LIN {X 0,Y 524.222,Z 576.731,A -85,B 0,C 180,E1 -4783.371,E2 -4783.371} C_VEL
LIN {X 0,Y 524.644,Z 566.022,A -85,B 0,C 180,E1 -4784.886,E2 -4784.886} C_VEL
LIN {X 0,Y 525.141,Z 554.055,A -85,B 0,C 180,E1 -4786.323,E2 -4786.323} C_VEL
LIN {X 0,Y 525.695,Z 541.49,A -85,B 0,C 180,E1 -4787.606,E2 -4787.606} C_VEL
LIN {X 0,Y 526.345,Z 527.816,A -85,B 0,C 180,E1 -4788.792,E2 -4788.792} C_VEL
LIN {X 0,Y 526.961,Z 514.228,A -85,B 0,C 180,E1 -4789.781,E2 -4789.781} C_VEL
LIN {X 0,Y 527.519,Z 499.628,A -85,B 0,C 180,E1 -4790.674,E2 -4790.674} C_VEL
LIN {X 0,Y 528.182,Z 483.147,A -85,B 0,C 180,E1 -4791.492,E2 -4791.492} C_VEL
LIN {X 0,Y 528.713,Z 467.343,A -85,B 0,C 180,E1 -4792.108,E2 -4792.108} C_VEL
LIN {X 0,Y 529.094,Z 451.309,A -85,B 0,C 180,E1 -4792.579,E2 -4792.579} C_VEL
LIN {X 0,Y 529.403,Z 434.816,A -85,B 0,C 180,E1 -4792.9,E2 -4792.9} C_VEL
LIN {X 0,Y 530.91,Z 248.916,A -85,B 0,C 180,E1 -4795.546,E2 -4795.546} C_VEL
LIN {X 0,Y 528.192,Z 233.834,A -85,B 0,C 180,E1 -4795.919,E2 -4795.919} C_VEL
LIN {X 0,Y 529.034,Z 209.98,A -85,B 0,C 180,E1 -4798.169,E2 -4798.169} C_VEL
LIN {X 0,Y 524.534,Z 194.611,A -85,B 0,C 180,E1 -4799.94,E2 -4799.94} C_VEL
LIN {X 0,Y 523.914,Z 192.537,A -85,B 0,C 180,E1 -4800.201,E2 -4800.201} C_VEL
LIN {X 0,Y 523.939,Z 192.528,A -85,B 0,C 180,E1 -4803.364,E2 -4803.364} C_VEL
LIN {X 0,Y 523.896,Z 192.537,A -85,B 0,C 180,E1 -4806.4,E2 -4806.4} C_VEL
LIN {X 0,Y 523.917,Z 192.54,A -85,B 0,C 180,E1 -4809.085,E2 -4809.085} C_VEL
LIN {X 0,Y 523.936,Z 192.53,A -85,B 0,C 180,E1 -4812.12,E2 -4812.12} C_VEL
LIN {X 0,Y 523.936,Z 192.531,A -85,B 0,C 180,E1 -4815.311,E2 -4815.311} C_VEL
LIN {X 0,Y 523.95,Z 192.533,A -85,B 0,C 180,E1 -4818.69,E2 -4818.69} C_VEL
LIN {X 0,Y 523.911,Z 192.533,A -85,B 0,C 180,E1 -4821.898,E2 -4821.898} C_VEL
LIN {X 0,Y 523.92,Z 192.537,A -85,B 0,C 180,E1 -4824.911,E2 -4824.911} C_VEL
LIN {X 0,Y 523.931,Z 192.526,A -85,B 0,C 180,E1 -4827.68,E2 -4827.68} C_VEL
LIN {X 0,Y 523.949,Z 192.534,A -85,B 0,C 180,E1 -4830.677,E2 -4830.677} C_VEL
LIN {X 0,Y 523.969,Z 192.519,A -85,B 0,C 180,E1 -4833.728,E2 -4833.728} C_VEL
LIN {X 0,Y 523.909,Z 192.534,A -85,B 0,C 180,E1 -4836.27,E2 -4836.27} C_VEL
LIN {X 0,Y 523.941,Z 192.531,A -85,B 0,C 180,E1 -4838.767,E2 -4838.767} C_VEL
LIN {X 0,Y 523.936,Z 192.524,A -85,B 0,C 180,E1 -4841.22,E2 -4841.22} C_VEL
LIN {X 0,Y 523.924,Z 192.53,A -85,B 0,C 180,E1 -4843.639,E2 -4843.639} C_VEL
LIN {X 0,Y 523.934,Z 192.531,A -85,B 0,C 180,E1 -4846.028,E2 -4846.028} C_VEL
LIN {X 0,Y 524.009,Z 192.516,A -85,B 0,C 180,E1 -4848.394,E2 -4848.394} C_VEL
LIN {X 0,Y 523.986,Z 192.522,A -85,B 0,C 180,E1 -4851.516,E2 -4851.516} C_VEL
LIN {X 0,Y 524.032,Z 192.519,A -85,B 0,C 180,E1 -4853.841,E2 -4853.841} C_VEL
LIN {X 0,Y 524.067,Z 192.501,A -85,B 0,C 180,E1 -4856.925,E2 -4856.925} C_VEL
LIN {X 0,Y 524.109,Z 192.509,A -85,B 0,C 180,E1 -4860,E2 -4860} C_VEL
LIN {X 0,Y 524.068,Z 192.511,A -85,B 0,C 180,E1 -4863.075,E2 -4863.075} C_VEL
LIN {X 0,Y 524.041,Z 192.518,A -85,B 0,C 180,E1 -4866.159,E2 -4866.159} C_VEL
LIN {X 0,Y 523.997,Z 192.525,A -85,B 0,C 180,E1 -4868.484,E2 -4868.484} C_VEL
LIN {X 0,Y 523.999,Z 192.521,A -85,B 0,C 180,E1 -4871.739,E2 -4871.739} C_VEL
LIN {X 0,Y 523.99,Z 192.522,A -85,B 0,C 180,E1 -4875.052,E2 -4875.052} C_VEL
LIN {X 0,Y 523.962,Z 192.527,A -85,B 0,C 180,E1 -4877.969,E2 -4877.969} C_VEL
LIN {X 0,Y 523.969,Z 192.526,A -85,B 0,C 180,E1 -4880.41,E2 -4880.41} C_VEL
LIN {X 0,Y 523.914,Z 192.531,A -85,B 0,C 180,E1 -4882.893,E2 -4882.893} C_VEL
LIN {X 0,Y 523.95,Z 192.525,A -85,B 0,C 180,E1 -4885.419,E2 -4885.419} C_VEL
LIN {X 0,Y 523.968,Z 192.531,A -85,B 0,C 180,E1 -4887.999,E2 -4887.999} C_VEL
LIN {X 0,Y 523.947,Z 192.525,A -85,B 0,C 180,E1 -4890.856,E2 -4890.856} C_VEL
LIN {X 0,Y 523.959,Z 192.532,A -85,B 0,C 180,E1 -4893.735,E2 -4893.735} C_VEL
LIN {X 0,Y 523.92,Z 192.53,A -85,B 0,C 180,E1 -4896.404,E2 -4896.404} C_VEL
LIN {X 0,Y 523.917,Z 192.529,A -85,B 0,C 180,E1 -4899.085,E2 -4899.085} C_VEL
LIN {X 0,Y 523.952,Z 192.527,A -85,B 0,C 180,E1 -4902.119,E2 -4902.119} C_VEL
LIN {X 0,Y 523.944,Z 192.531,A -85,B 0,C 180,E1 -4905.31,E2 -4905.31} C_VEL
LIN {X 0,Y 523.916,Z 192.533,A -85,B 0,C 180,E1 -4906.916,E2 -4906.916} C_VEL
LIN {X 0,Y 523.249,Z 192.62,A -85,B 0,C 180,E1 -4907.558,E2 -4907.558} C_VEL
LIN {X 0,Y 520.407,Z 192.971,A -85,B 0,C 180,E1 -4908.599,E2 -4908.599} C_VEL
LIN {X 0,Y 518.003,Z 193.272,A -85,B 0,C 180,E1 -4909.438,E2 -4909.438} C_VEL
LIN {X 0,Y 516.966,Z 193.398,A -85,B 0,C 180,E1 -4910.086,E2 -4910.086} C_VEL
LIN {X 0,Y 516.879,Z 193.408,A -85,B 0,C 180,E1 -4910.305,E2 -4910.305} C_VEL
LIN {X 0,Y 516.875,Z 193.412,A -85,B 0,C 180,E1 -4913.343,E2 -4913.343} C_VEL
LIN {X 0,Y 516.909,Z 193.406,A -85,B 0,C 180,E1 -4916.121,E2 -4916.121} C_VEL
LIN {X 0,Y 516.89,Z 193.408,A -85,B 0,C 180,E1 -4918.936,E2 -4918.936} C_VEL
LIN {X 0,Y 516.917,Z 193.406,A -85,B 0,C 180,E1 -4921.585,E2 -4921.585} C_VEL
LIN {X 0,Y 516.931,Z 193.402,A -85,B 0,C 180,E1 -4924.211,E2 -4924.211} C_VEL
LIN {X 0,Y 516.865,Z 193.411,A -85,B 0,C 180,E1 -4926.776,E2 -4926.776} C_VEL
LIN {X 0,Y 516.939,Z 193.397,A -85,B 0,C 180,E1 -4929.732,E2 -4929.732} C_VEL
LIN {X 0,Y 516.906,Z 193.405,A -85,B 0,C 180,E1 -4932.595,E2 -4932.595} C_VEL
LIN {X 0,Y 516.942,Z 193.402,A -85,B 0,C 180,E1 -4935.03,E2 -4935.03} C_VEL
LIN {X 0,Y 516.965,Z 193.4,A -85,B 0,C 180,E1 -4938.234,E2 -4938.234} C_VEL
LIN {X 0,Y 516.968,Z 193.402,A -85,B 0,C 180,E1 -4941.4,E2 -4941.4} C_VEL
LIN {X 0,Y 517.026,Z 193.393,A -85,B 0,C 180,E1 -4944.54,E2 -4944.54} C_VEL
LIN {X 0,Y 517.047,Z 193.434,A -85,B 0,C 180,E1 -4947.979,E2 -4947.979} C_VEL
LIN {X 0,Y 520.935,Z 207.525,A -85,B 0,C 180,E1 -4949.764,E2 -4949.764} C_VEL
LIN {X 0,Y 522.633,Z 212.295,A -85,B 0,C 180,E1 -4949.929,E2 -4949.929} C_VEL
LIN {X 0,Y 524.563,Z 222.327,A -85,B 0,C 180,E1 -4950.184,E2 -4950.184} C_VEL
LIN {X 0,Y 522.855,Z 413.311,A -85,B 0,C 180,E1 -4952.961,E2 -4952.961} C_VEL
LIN {X 0,Y 522.525,Z 429.48,A -85,B 0,C 180,E1 -4953.349,E2 -4953.349} C_VEL
LIN {X 0,Y 521.977,Z 445.854,A -85,B 0,C 180,E1 -4953.898,E2 -4953.898} C_VEL
LIN {X 0,Y 521.414,Z 460.885,A -85,B 0,C 180,E1 -4954.555,E2 -4954.555} C_VEL
LIN {X 0,Y 520.78,Z 476.68,A -85,B 0,C 180,E1 -4955.42,E2 -4955.42} C_VEL
LIN {X 0,Y 520.083,Z 491.283,A -85,B 0,C 180,E1 -4956.401,E2 -4956.401} C_VEL
LIN {X 0,Y 519.44,Z 504.752,A -85,B 0,C 180,E1 -4957.482,E2 -4957.482} C_VEL
LIN {X 0,Y 518.713,Z 518.29,A -85,B 0,C 180,E1 -4958.767,E2 -4958.767} C_VEL
LIN {X 0,Y 518.081,Z 530.647,A -85,B 0,C 180,E1 -4960.157,E2 -4960.157} C_VEL
LIN {X 0,Y 517.589,Z 541.233,A -85,B 0,C 180,E1 -4961.553,E2 -4961.553} C_VEL
LIN {X 0,Y 517.153,Z 551.508,A -85,B 0,C 180,E1 -4963.157,E2 -4963.157} C_VEL
LIN {X 0,Y 516.805,Z 560.149,A -85,B 0,C 180,E1 -4964.772,E2 -4964.772} C_VEL
LIN {X 0,Y 516.566,Z 566.583,A -85,B 0,C 180,E1 -4966.195,E2 -4966.195} C_VEL
LIN {X 0,Y 516.446,Z 572.319,A -85,B 0,C 180,E1 -4967.715,E2 -4967.715} C_VEL
LIN {X 0,Y 516.32,Z 577.625,A -85,B 0,C 180,E1 -4969.48,E2 -4969.48} C_VEL
LIN {X 0,Y 516.228,Z 580.6,A -85,B 0,C 180,E1 -4970.73,E2 -4970.73} C_VEL
LIN {X 0,Y 516.174,Z 583.527,A -85,B 0,C 180,E1 -4972.41,E2 -4972.41} C_VEL
LIN {X 0,Y 516.138,Z 585.436,A -85,B 0,C 180,E1 -4974.174,E2 -4974.174} C_VEL
LIN {X 0,Y 516.146,Z 586.138,A -85,B 0,C 180,E1 -4976.016,E2 -4976.016} C_VEL
LIN {X 0,Y 516.168,Z 585.538,A -85,B 0,C 180,E1 -4977.746,E2 -4977.746} C_VEL
LIN {X 0,Y 516.193,Z 583.95,A -85,B 0,C 180,E1 -4979.383,E2 -4979.383} C_VEL
LIN {X 0,Y 516.235,Z 581.052,A -85,B 0,C 180,E1 -4981.153,E2 -4981.153} C_VEL
LIN {X 0,Y 516.314,Z 578.077,A -85,B 0,C 180,E1 -4982.442,E2 -4982.442} C_VEL
LIN {X 0,Y 516.384,Z 573.835,A -85,B 0,C 180,E1 -4983.918,E2 -4983.918} C_VEL
LIN {X 0,Y 516.54,Z 568.152,A -85,B 0,C 180,E1 -4985.508,E2 -4985.508} C_VEL
LIN {X 0,Y 516.737,Z 560.548,A -85,B 0,C 180,E1 -4987.245,E2 -4987.245} C_VEL
LIN {X 0,Y 517.046,Z 552.873,A -85,B 0,C 180,E1 -4988.7,E2 -4988.7} C_VEL
LIN {X 0,Y 517.441,Z 543.71,A -85,B 0,C 180,E1 -4990.176,E2 -4990.176} C_VEL
LIN {X 0,Y 517.976,Z 532.31,A -85,B 0,C 180,E1 -4991.734,E2 -4991.734} C_VEL
LIN {X 0,Y 518.636,Z 519.838,A -85,B 0,C 180,E1 -4993.168,E2 -4993.168} C_VEL
LIN {X 0,Y 519.267,Z 507.368,A -85,B 0,C 180,E1 -4994.388,E2 -4994.388} C_VEL
LIN {X 0,Y 520.016,Z 492.6,A -85,B 0,C 180,E1 -4995.6,E2 -4995.6} C_VEL
LIN {X 0,Y 520.798,Z 476.677,A -85,B 0,C 180,E1 -4996.675,E2 -4996.675} C_VEL
LIN {X 0,Y 521.453,Z 460.886,A -85,B 0,C 180,E1 -4997.538,E2 -4997.538} C_VEL
LIN {X 0,Y 522.01,Z 445.593,A -85,B 0,C 180,E1 -4998.204,E2 -4998.204} C_VEL
LIN {X 0,Y 522.498,Z 429.104,A -85,B 0,C 180,E1 -4998.754,E2 -4998.754} C_VEL
LIN {X 0,Y 522.873,Z 412.973,A -85,B 0,C 180,E1 -4999.135,E2 -4999.135} C_VEL
LIN {X 0,Y 524.555,Z 221.705,A -85,B 0,C 180,E1 -5001.919,E2 -5001.919} C_VEL
LIN {X 0,Y 522.049,Z 210.335,A -85,B 0,C 180,E1 -5002.227,E2 -5002.227} C_VEL
LIN {X 0,Y 520.799,Z 207.327,A -85,B 0,C 180,E1 -5002.365,E2 -5002.365} C_VEL
LIN {X 0,Y 516.875,Z 193.415,A -85,B 0,C 180,E1 -5004.19,E2 -5004.19} C_VEL
LIN {X 0,Y 516.874,Z 193.417,A -85,B 0,C 180,E1 -5007.052,E2 -5007.052} C_VEL
LIN {X 0,Y 516.875,Z 193.413,A -85,B 0,C 180,E1 -5009.795,E2 -5009.795} C_VEL
LIN {X 0,Y 516.883,Z 193.412,A -85,B 0,C 180,E1 -5012.465,E2 -5012.465} C_VEL
LIN {X 0,Y 516.866,Z 193.412,A -85,B 0,C 180,E1 -5015.645,E2 -5015.645} C_VEL
LIN {X 0,Y 516.877,Z 193.41,A -85,B 0,C 180,E1 -5018.462,E2 -5018.462} C_VEL
LIN {X 0,Y 516.892,Z 193.411,A -85,B 0,C 180,E1 -5020.955,E2 -5020.955} C_VEL
LIN {X 0,Y 516.897,Z 193.407,A -85,B 0,C 180,E1 -5023.41,E2 -5023.41} C_VEL
LIN {X 0,Y 516.885,Z 193.409,A -85,B 0,C 180,E1 -5025.833,E2 -5025.833} C_VEL
LIN {X 0,Y 516.958,Z 193.399,A -85,B 0,C 180,E1 -5028.234,E2 -5028.234} C_VEL
LIN {X 0,Y 516.95,Z 193.4,A -85,B 0,C 180,E1 -5031.399,E2 -5031.399} C_VEL
LIN {X 0,Y 516.994,Z 193.394,A -85,B 0,C 180,E1 -5033.757,E2 -5033.757} C_VEL
LIN {X 0,Y 517.006,Z 193.395,A -85,B 0,C 180,E1 -5036.883,E2 -5036.883} C_VEL
LIN {X 0,Y 517.076,Z 193.389,A -85,B 0,C 180,E1 -5040,E2 -5040} C_VEL
LIN {X 0,Y 517.006,Z 193.391,A -85,B 0,C 180,E1 -5043.117,E2 -5043.117} C_VEL
LIN {X 0,Y 517.002,Z 193.4,A -85,B 0,C 180,E1 -5046.243,E2 -5046.243} C_VEL
LIN {X 0,Y 516.948,Z 193.401,A -85,B 0,C 180,E1 -5049.389,E2 -5049.389} C_VEL
LIN {X 0,Y 516.945,Z 193.404,A -85,B 0,C 180,E1 -5051.808,E2 -5051.808} C_VEL
LIN {X 0,Y 516.937,Z 193.402,A -85,B 0,C 180,E1 -5055.147,E2 -5055.147} C_VEL
LIN {X 0,Y 516.919,Z 193.406,A -85,B 0,C 180,E1 -5058.222,E2 -5058.222} C_VEL
LIN {X 0,Y 516.906,Z 193.406,A -85,B 0,C 180,E1 -5060.702,E2 -5060.702} C_VEL
LIN {X 0,Y 516.905,Z 193.409,A -85,B 0,C 180,E1 -5064.072,E2 -5064.072} C_VEL
LIN {X 0,Y 516.923,Z 193.402,A -85,B 0,C 180,E1 -5066.658,E2 -5066.658} C_VEL
LIN {X 0,Y 516.905,Z 193.412,A -85,B 0,C 180,E1 -5069.524,E2 -5069.524} C_VEL
LIN {X 0,Y 516.895,Z 193.408,A -85,B 0,C 180,E1 -5072.545,E2 -5072.545} C_VEL
LIN {X 0,Y 516.865,Z 193.42,A -85,B 0,C 180,E1 -5075.331,E2 -5075.331} C_VEL
LIN {X 0,Y 516.875,Z 193.413,A -85,B 0,C 180,E1 -5077.944,E2 -5077.944} C_VEL
LIN {X 0,Y 516.879,Z 193.413,A -85,B 0,C 180,E1 -5080.742,E2 -5080.742} C_VEL
LIN {X 0,Y 516.878,Z 193.415,A -85,B 0,C 180,E1 -5082.832,E2 -5082.832} C_VEL
LIN {X 0,Y 516.918,Z 193.414,A -85,B 0,C 180,E1 -5085.011,E2 -5085.011} C_VEL
LIN {X 0,Y 516.908,Z 193.409,A -85,B 0,C 180,E1 -5088.399,E2 -5088.399} C_VEL
LIN {X 0,Y 516.877,Z 193.414,A -85,B 0,C 180,E1 -5091.285,E2 -5091.285} C_VEL
LIN {X 0,Y 516.866,Z 193.414,A -85,B 0,C 180,E1 -5094.22,E2 -5094.22} C_VEL
LIN {X 0,Y 516.891,Z 193.416,A -85,B 0,C 180,E1 -5097.053,E2 -5097.053} C_VEL
LIN {X 0,Y 516.916,Z 193.581,A -85,B 0,C 180,E1 -5099.516,E2 -5099.516} C_VEL
LIN {X 0,Y 522.209,Z 211.448,A -85,B 0,C 180,E1 -5101.62,E2 -5101.62} C_VEL
LIN {X 0,Y 521.508,Z 233.414,A -85,B 0,C 180,E1 -5103.727,E2 -5103.727} C_VEL
LIN {X 0,Y 524.478,Z 250.636,A -85,B 0,C 180,E1 -5104.151,E2 -5104.151} C_VEL
LIN {X 0,Y 522.789,Z 438.701,A -85,B 0,C 180,E1 -5106.872,E2 -5106.872} C_VEL
LIN {X 0,Y 522.446,Z 454.476,A -85,B 0,C 180,E1 -5107.222,E2 -5107.222} C_VEL
LIN {X 0,Y 522.001,Z 469.792,A -85,B 0,C 180,E1 -5107.698,E2 -5107.698} C_VEL
LIN {X 0,Y 521.425,Z 484.424,A -85,B 0,C 180,E1 -5108.294,E2 -5108.294} C_VEL
LIN {X 0,Y 520.852,Z 499.253,A -85,B 0,C 180,E1 -5109.049,E2 -5109.049} C_VEL
LIN {X 0,Y 520.249,Z 512.438,A -85,B 0,C 180,E1 -5109.851,E2 -5109.851} C_VEL
LIN {X 0,Y 519.508,Z 527.483,A -85,B 0,C 180,E1 -5110.952,E2 -5110.952} C_VEL
LIN {X 0,Y 518.864,Z 540.105,A -85,B 0,C 180,E1 -5112.053,E2 -5112.053} C_VEL
LIN {X 0,Y 518.276,Z 551.972,A -85,B 0,C 180,E1 -5113.253,E2 -5113.253} C_VEL
LIN {X 0,Y 517.734,Z 563.934,A -85,B 0,C 180,E1 -5114.666,E2 -5114.666} C_VEL
LIN {X 0,Y 517.265,Z 575.232,A -85,B 0,C 180,E1 -5116.245,E2 -5116.245} C_VEL
LIN {X 0,Y 516.933,Z 584.758,A -85,B 0,C 180,E1 -5117.835,E2 -5117.835} C_VEL
LIN {X 0,Y 516.672,Z 592.73,A -85,B 0,C 180,E1 -5119.419,E2 -5119.419} C_VEL
LIN {X 0,Y 516.468,Z 599.381,A -85,B 0,C 180,E1 -5120.997,E2 -5120.997} C_VEL
LIN {X 0,Y 516.371,Z 604.775,A -85,B 0,C 180,E1 -5122.571,E2 -5122.571} C_VEL
LIN {X 0,Y 516.319,Z 608.108,A -85,B 0,C 180,E1 -5123.749,E2 -5123.749} C_VEL
LIN {X 0,Y 516.225,Z 611.529,A -85,B 0,C 180,E1 -5125.315,E2 -5125.315} C_VEL
LIN {X 0,Y 516.267,Z 614.018,A -85,B 0,C 180,E1 -5126.879,E2 -5126.879} C_VEL
LIN {X 0,Y 516.186,Z 615.418,A -85,B 0,C 180,E1 -5128.44,E2 -5128.44} C_VEL
LIN {X 0,Y 516.149,Z 615.946,A -85,B 0,C 180,E1 -5130,E2 -5130} C_VEL
LIN {X 0,Y 516.186,Z 615.418,A -85,B 0,C 180,E1 -5131.561,E2 -5131.561} C_VEL
LIN {X 0,Y 516.267,Z 614.017,A -85,B 0,C 180,E1 -5133.122,E2 -5133.122} C_VEL
LIN {X 0,Y 516.225,Z 611.53,A -85,B 0,C 180,E1 -5134.686,E2 -5134.686} C_VEL
LIN {X 0,Y 516.368,Z 607.414,A -85,B 0,C 180,E1 -5136.507,E2 -5136.507} C_VEL
LIN {X 0,Y 516.418,Z 602.265,A -85,B 0,C 180,E1 -5138.216,E2 -5138.216} C_VEL
LIN {X 0,Y 516.591,Z 594.571,A -85,B 0,C 180,E1 -5140.187,E2 -5140.187} C_VEL
LIN {X 0,Y 516.904,Z 585.889,A -85,B 0,C 180,E1 -5141.967,E2 -5141.967} C_VEL
LIN {X 0,Y 517.203,Z 576.513,A -85,B 0,C 180,E1 -5143.556,E2 -5143.556} C_VEL
LIN {X 0,Y 517.635,Z 566.866,A -85,B 0,C 180,E1 -5144.949,E2 -5144.949} C_VEL
LIN {X 0,Y 518.134,Z 555.623,A -85,B 0,C 180,E1 -5146.347,E2 -5146.347} C_VEL
LIN {X 0,Y 518.751,Z 543.377,A -85,B 0,C 180,E1 -5147.646,E2 -5147.646} C_VEL
LIN {X 0,Y 519.397,Z 530.405,A -85,B 0,C 180,E1 -5148.812,E2 -5148.812} C_VEL
LIN {X 0,Y 520.043,Z 516.853,A -85,B 0,C 180,E1 -5149.849,E2 -5149.849} C_VEL
LIN {X 0,Y 520.639,Z 502.921,A -85,B 0,C 180,E1 -5150.753,E2 -5150.753} C_VEL
LIN {X 0,Y 521.415,Z 487.208,A -85,B 0,C 180,E1 -5151.584,E2 -5151.584} C_VEL
LIN {X 0,Y 521.956,Z 471.272,A -85,B 0,C 180,E1 -5152.253,E2 -5152.253} C_VEL
LIN {X 0,Y 522.403,Z 455.599,A -85,B 0,C 180,E1 -5152.754,E2 -5152.754} C_VEL
LIN {X 0,Y 522.791,Z 438.955,A -85,B 0,C 180,E1 -5153.128,E2 -5153.128} C_VEL
LIN {X 0,Y 524.44,Z 249.524,A -85,B 0,C 180,E1 -5155.872,E2 -5155.872} C_VEL
LIN {X 0,Y 521.559,Z 233.731,A -85,B 0,C 180,E1 -5156.265,E2 -5156.265} C_VEL
LIN {X 0,Y 522.325,Z 211.669,A -85,B 0,C 180,E1 -5158.379,E2 -5158.379} C_VEL
LIN {X 0,Y 516.901,Z 193.409,A -85,B 0,C 180,E1 -5160.542,E2 -5160.542} C_VEL
LIN {X 0,Y 516.892,Z 193.401,A -85,B 0,C 180,E1 -5162.947,E2 -5162.947} C_VEL
LIN {X 0,Y 516.865,Z 193.415,A -85,B 0,C 180,E1 -5165.781,E2 -5165.781} C_VEL
LIN {X 0,Y 516.877,Z 193.414,A -85,B 0,C 180,E1 -5168.716,E2 -5168.716} C_VEL
LIN {X 0,Y 516.899,Z 193.408,A -85,B 0,C 180,E1 -5171.776,E2 -5171.776} C_VEL
LIN {X 0,Y 516.892,Z 193.412,A -85,B 0,C 180,E1 -5175.007,E2 -5175.007} C_VEL
LIN {X 0,Y 516.906,Z 193.408,A -85,B 0,C 180,E1 -5178.399,E2 -5178.399} C_VEL
LIN {X 0,Y 516.874,Z 193.414,A -85,B 0,C 180,E1 -5181.284,E2 -5181.284} C_VEL
LIN {X 0,Y 516.867,Z 193.406,A -85,B 0,C 180,E1 -5184.22,E2 -5184.22} C_VEL
LIN {X 0,Y 516.878,Z 193.41,A -85,B 0,C 180,E1 -5187.052,E2 -5187.052} C_VEL
LIN {X 0,Y 516.888,Z 193.406,A -85,B 0,C 180,E1 -5189.796,E2 -5189.796} C_VEL
LIN {X 0,Y 516.92,Z 193.409,A -85,B 0,C 180,E1 -5192.467,E2 -5192.467} C_VEL
LIN {X 0,Y 516.869,Z 193.412,A -85,B 0,C 180,E1 -5195.07,E2 -5195.07} C_VEL
LIN {X 0,Y 516.865,Z 193.411,A -85,B 0,C 180,E1 -5197.621,E2 -5197.621} C_VEL
LIN {X 0,Y 516.926,Z 193.4,A -85,B 0,C 180,E1 -5200.13,E2 -5200.13} C_VEL
LIN {X 0,Y 516.893,Z 193.41,A -85,B 0,C 180,E1 -5202.595,E2 -5202.595} C_VEL
LIN {X 0,Y 516.939,Z 193.402,A -85,B 0,C 180,E1 -5205.03,E2 -5205.03} C_VEL
LIN {X 0,Y 516.962,Z 193.393,A -85,B 0,C 180,E1 -5208.234,E2 -5208.234} C_VEL
LIN {X 0,Y 516.954,Z 193.398,A -85,B 0,C 180,E1 -5211.399,E2 -5211.399} C_VEL
LIN {X 0,Y 516.998,Z 193.394,A -85,B 0,C 180,E1 -5213.757,E2 -5213.757} C_VEL
LIN {X 0,Y 517.008,Z 193.38,A -85,B 0,C 180,E1 -5216.883,E2 -5216.883} C_VEL
LIN {X 0,Y 517.08,Z 193.384,A -85,B 0,C 180,E1 -5220,E2 -5220} C_VEL
LIN {X 0,Y 517.008,Z 193.391,A -85,B 0,C 180,E1 -5223.117,E2 -5223.117} C_VEL
LIN {X 0,Y 517.005,Z 193.395,A -85,B 0,C 180,E1 -5226.243,E2 -5226.243} C_VEL
LIN {X 0,Y 516.942,Z 193.401,A -85,B 0,C 180,E1 -5229.389,E2 -5229.389} C_VEL
LIN {X 0,Y 516.949,Z 193.399,A -85,B 0,C 180,E1 -5231.807,E2 -5231.807} C_VEL
LIN {X 0,Y 516.941,Z 193.4,A -85,B 0,C 180,E1 -5235.146,E2 -5235.146} C_VEL
LIN {X 0,Y 516.923,Z 193.4,A -85,B 0,C 180,E1 -5238.222,E2 -5238.222} C_VEL
LIN {X 0,Y 516.909,Z 193.404,A -85,B 0,C 180,E1 -5240.702,E2 -5240.702} C_VEL
LIN {X 0,Y 516.909,Z 193.405,A -85,B 0,C 180,E1 -5244.072,E2 -5244.072} C_VEL
LIN {X 0,Y 516.924,Z 193.4,A -85,B 0,C 180,E1 -5246.658,E2 -5246.658} C_VEL
LIN {X 0,Y 516.917,Z 193.409,A -85,B 0,C 180,E1 -5249.526,E2 -5249.526} C_VEL
LIN {X 0,Y 516.895,Z 193.402,A -85,B 0,C 180,E1 -5252.544,E2 -5252.544} C_VEL
LIN {X 0,Y 516.881,Z 193.412,A -85,B 0,C 180,E1 -5255.332,E2 -5255.332} C_VEL
LIN {X 0,Y 516.878,Z 193.408,A -85,B 0,C 180,E1 -5257.943,E2 -5257.943} C_VEL
LIN {X 0,Y 516.882,Z 193.408,A -85,B 0,C 180,E1 -5260.742,E2 -5260.742} C_VEL
LIN {X 0,Y 516.88,Z 193.407,A -85,B 0,C 180,E1 -5262.832,E2 -5262.832} C_VEL
LIN {X 0,Y 516.88,Z 193.41,A -85,B 0,C 180,E1 -5266.097,E2 -5266.097} C_VEL
LIN {X 0,Y 516.911,Z 193.401,A -85,B 0,C 180,E1 -5268.399,E2 -5268.399} C_VEL
LIN {X 0,Y 516.879,Z 193.408,A -85,B 0,C 180,E1 -5270.305,E2 -5270.305} C_VEL
LIN {X 0,Y 516.208,Z 193.495,A -85,B 0,C 180,E1 -5270.956,E2 -5270.956} C_VEL
LIN {X 0,Y 513.36,Z 193.851,A -85,B 0,C 180,E1 -5272.011,E2 -5272.011} C_VEL
LIN {X 0,Y 510.95,Z 194.152,A -85,B 0,C 180,E1 -5272.861,E2 -5272.861} C_VEL
LIN {X 0,Y 509.908,Z 194.278,A -85,B 0,C 180,E1 -5273.518,E2 -5273.518} C_VEL
LIN {X 0,Y 509.819,Z 194.287,A -85,B 0,C 180,E1 -5273.74,E2 -5273.74} C_VEL
LIN {X 0,Y 509.859,Z 194.284,A -85,B 0,C 180,E1 -5276.539,E2 -5276.539} C_VEL
LIN {X 0,Y 509.844,Z 194.289,A -85,B 0,C 180,E1 -5279.334,E2 -5279.334} C_VEL
LIN {X 0,Y 509.891,Z 194.277,A -85,B 0,C 180,E1 -5282.055,E2 -5282.055} C_VEL
LIN {X 0,Y 509.875,Z 194.284,A -85,B 0,C 180,E1 -5284.704,E2 -5284.704} C_VEL
LIN {X 0,Y 509.826,Z 194.293,A -85,B 0,C 180,E1 -5287.458,E2 -5287.458} C_VEL
LIN {X 0,Y 509.916,Z 194.271,A -85,B 0,C 180,E1 -5289.845,E2 -5289.845} C_VEL
LIN {X 0,Y 509.873,Z 194.29,A -85,B 0,C 180,E1 -5293.174,E2 -5293.174} C_VEL
LIN {X 0,Y 509.863,Z 194.275,A -85,B 0,C 180,E1 -5295.634,E2 -5295.634} C_VEL
LIN {X 0,Y 509.913,Z 194.283,A -85,B 0,C 180,E1 -5298.874,E2 -5298.874} C_VEL
LIN {X 0,Y 509.951,Z 194.274,A -85,B 0,C 180,E1 -5302.078,E2 -5302.078} C_VEL
LIN {X 0,Y 509.977,Z 194.27,A -85,B 0,C 180,E1 -5304.464,E2 -5304.464} C_VEL
LIN {X 0,Y 510.06,Z 194.433,A -85,B 0,C 180,E1 -5307.655,E2 -5307.655} C_VEL
LIN {X 0,Y 513.763,Z 207.706,A -85,B 0,C 180,E1 -5309.369,E2 -5309.369} C_VEL
LIN {X 0,Y 516.386,Z 214.022,A -85,B 0,C 180,E1 -5309.613,E2 -5309.613} C_VEL
LIN {X 0,Y 518.206,Z 223.729,A -85,B 0,C 180,E1 -5309.862,E2 -5309.862} C_VEL
LIN {X 0,Y 516.32,Z 413.641,A -85,B 0,C 180,E1 -5312.657,E2 -5312.657} C_VEL
LIN {X 0,Y 515.963,Z 429.736,A -85,B 0,C 180,E1 -5313.05,E2 -5313.05} C_VEL
LIN {X 0,Y 515.445,Z 445.07,A -85,B 0,C 180,E1 -5313.566,E2 -5313.566} C_VEL
LIN {X 0,Y 514.831,Z 460.426,A -85,B 0,C 180,E1 -5314.235,E2 -5314.235} C_VEL
LIN {X 0,Y 514.142,Z 476.124,A -85,B 0,C 180,E1 -5315.097,E2 -5315.097} C_VEL
LIN {X 0,Y 513.37,Z 490.867,A -85,B 0,C 180,E1 -5316.09,E2 -5316.09} C_VEL
LIN {X 0,Y 512.663,Z 504.439,A -85,B 0,C 180,E1 -5317.186,E2 -5317.186} C_VEL
LIN {X 0,Y 511.938,Z 517.566,A -85,B 0,C 180,E1 -5318.437,E2 -5318.437} C_VEL
LIN {X 0,Y 511.285,Z 528.87,A -85,B 0,C 180,E1 -5319.694,E2 -5319.694} C_VEL
LIN {X 0,Y 510.706,Z 539.691,A -85,B 0,C 180,E1 -5321.108,E2 -5321.108} C_VEL
LIN {X 0,Y 510.297,Z 548.976,A -85,B 0,C 180,E1 -5322.526,E2 -5322.526} C_VEL
LIN {X 0,Y 509.85,Z 558.103,A -85,B 0,C 180,E1 -5324.162,E2 -5324.162} C_VEL
LIN {X 0,Y 509.604,Z 564.851,A -85,B 0,C 180,E1 -5325.6,E2 -5325.6} C_VEL
LIN {X 0,Y 509.41,Z 571.312,A -85,B 0,C 180,E1 -5327.254,E2 -5327.254} C_VEL
LIN {X 0,Y 509.27,Z 576.596,A -85,B 0,C 180,E1 -5328.923,E2 -5328.923} C_VEL
LIN {X 0,Y 509.203,Z 579.78,A -85,B 0,C 180,E1 -5330.194,E2 -5330.194} C_VEL
LIN {X 0,Y 509.092,Z 583.064,A -85,B 0,C 180,E1 -5331.884,E2 -5331.884} C_VEL
LIN {X 0,Y 509.04,Z 585.178,A -85,B 0,C 180,E1 -5333.602,E2 -5333.602} C_VEL
LIN {X 0,Y 509.039,Z 586.211,A -85,B 0,C 180,E1 -5335.34,E2 -5335.34} C_VEL
LIN {X 0,Y 509.056,Z 586.135,A -85,B 0,C 180,E1 -5337.103,E2 -5337.103} C_VEL
LIN {X 0,Y 509.083,Z 584.783,A -85,B 0,C 180,E1 -5338.893,E2 -5338.893} C_VEL
LIN {X 0,Y 509.142,Z 582.179,A -85,B 0,C 180,E1 -5340.712,E2 -5340.712} C_VEL
LIN {X 0,Y 509.232,Z 579.347,A -85,B 0,C 180,E1 -5342.096,E2 -5342.096} C_VEL
LIN {X 0,Y 509.283,Z 575.644,A -85,B 0,C 180,E1 -5343.503,E2 -5343.503} C_VEL
LIN {X 0,Y 509.423,Z 571.015,A -85,B 0,C 180,E1 -5344.926,E2 -5344.926} C_VEL
LIN {X 0,Y 509.59,Z 564.262,A -85,B 0,C 180,E1 -5346.631,E2 -5346.631} C_VEL
LIN {X 0,Y 509.97,Z 556.074,A -85,B 0,C 180,E1 -5348.326,E2 -5348.326} C_VEL
LIN {X 0,Y 510.356,Z 547.084,A -85,B 0,C 180,E1 -5349.885,E2 -5349.885} C_VEL
LIN {X 0,Y 510.854,Z 537.25,A -85,B 0,C 180,E1 -5351.326,E2 -5351.326} C_VEL
LIN {X 0,Y 511.428,Z 526.115,A -85,B 0,C 180,E1 -5352.726,E2 -5352.726} C_VEL
LIN {X 0,Y 512.129,Z 514.206,A -85,B 0,C 180,E1 -5354.005,E2 -5354.005} C_VEL
LIN {X 0,Y 512.841,Z 501.432,A -85,B 0,C 180,E1 -5355.172,E2 -5355.172} C_VEL
LIN {X 0,Y 513.59,Z 487.425,A -85,B 0,C 180,E1 -5356.251,E2 -5356.251} C_VEL
LIN {X 0,Y 514.331,Z 471.983,A -85,B 0,C 180,E1 -5357.24,E2 -5357.24} C_VEL
LIN {X 0,Y 515.054,Z 456.539,A -85,B 0,C 180,E1 -5358.04,E2 -5358.04} C_VEL
LIN {X 0,Y 515.583,Z 441.015,A -85,B 0,C 180,E1 -5358.683,E2 -5358.683} C_VEL
LIN {X 0,Y 516.101,Z 423.885,A -85,B 0,C 180,E1 -5359.205,E2 -5359.205} C_VEL
LIN {X 0,Y 516.41,Z 406.886,A -85,B 0,C 180,E1 -5359.549,E2 -5359.549} C_VEL
LIN {X 0,Y 518.22,Z 223.432,A -85,B 0,C 180,E1 -5362.237,E2 -5362.237} C_VEL
LIN {X 0,Y 516.056,Z 213.161,A -85,B 0,C 180,E1 -5362.515,E2 -5362.515} C_VEL
LIN {X 0,Y 513.627,Z 207.57,A -85,B 0,C 180,E1 -5362.762,E2 -5362.762} C_VEL
LIN {X 0,Y 509.862,Z 194.289,A -85,B 0,C 180,E1 -5364.539,E2 -5364.539} C_VEL
LIN {X 0,Y 509.852,Z 194.29,A -85,B 0,C 180,E1 -5367.48,E2 -5367.48} C_VEL
LIN {X 0,Y 509.85,Z 194.288,A -85,B 0,C 180,E1 -5370.274,E2 -5370.274} C_VEL
LIN {X 0,Y 509.824,Z 194.292,A -85,B 0,C 180,E1 -5372.941,E2 -5372.941} C_VEL
LIN {X 0,Y 509.828,Z 194.289,A -85,B 0,C 180,E1 -5375.572,E2 -5375.572} C_VEL
LIN {X 0,Y 509.813,Z 194.287,A -85,B 0,C 180,E1 -5378.148,E2 -5378.148} C_VEL
LIN {X 0,Y 509.854,Z 194.288,A -85,B 0,C 180,E1 -5380.681,E2 -5380.681} C_VEL
LIN {X 0,Y 509.864,Z 194.285,A -85,B 0,C 180,E1 -5383.174,E2 -5383.174} C_VEL
LIN {X 0,Y 509.855,Z 194.284,A -85,B 0,C 180,E1 -5385.634,E2 -5385.634} C_VEL
LIN {X 0,Y 509.905,Z 194.283,A -85,B 0,C 180,E1 -5388.874,E2 -5388.874} C_VEL
LIN {X 0,Y 509.914,Z 194.279,A -85,B 0,C 180,E1 -5392.078,E2 -5392.078} C_VEL
LIN {X 0,Y 509.97,Z 194.278,A -85,B 0,C 180,E1 -5394.464,E2 -5394.464} C_VEL
LIN {X 0,Y 510.045,Z 194.261,A -85,B 0,C 180,E1 -5397.631,E2 -5397.631} C_VEL
LIN {X 0,Y 510.058,Z 194.261,A -85,B 0,C 180,E1 -5400.789,E2 -5400.789} C_VEL
LIN {X 0,Y 509.948,Z 194.27,A -85,B 0,C 180,E1 -5403.16,E2 -5403.16} C_VEL
LIN {X 0,Y 509.97,Z 194.276,A -85,B 0,C 180,E1 -5406.33,E2 -5406.33} C_VEL
LIN {X 0,Y 509.909,Z 194.278,A -85,B 0,C 180,E1 -5408.72,E2 -5408.72} C_VEL
LIN {X 0,Y 509.897,Z 194.284,A -85,B 0,C 180,E1 -5411.932,E2 -5411.932} C_VEL
LIN {X 0,Y 509.887,Z 194.281,A -85,B 0,C 180,E1 -5415.242,E2 -5415.242} C_VEL
LIN {X 0,Y 509.882,Z 194.286,A -85,B 0,C 180,E1 -5418.001,E2 -5418.001} C_VEL
LIN {X 0,Y 509.844,Z 194.286,A -85,B 0,C 180,E1 -5421.002,E2 -5421.002} C_VEL
LIN {X 0,Y 509.83,Z 194.294,A -85,B 0,C 180,E1 -5423.563,E2 -5423.563} C_VEL
LIN {X 0,Y 509.907,Z 194.276,A -85,B 0,C 180,E1 -5426.379,E2 -5426.379} C_VEL
LIN {X 0,Y 509.871,Z 194.283,A -85,B 0,C 180,E1 -5428.844,E2 -5428.844} C_VEL
LIN {X 0,Y 509.82,Z 194.295,A -85,B 0,C 180,E1 -5431.59,E2 -5431.59} C_VEL
LIN {X 0,Y 509.845,Z 194.287,A -85,B 0,C 180,E1 -5434.414,E2 -5434.414} C_VEL
LIN {X 0,Y 509.811,Z 194.299,A -85,B 0,C 180,E1 -5437.341,E2 -5437.341} C_VEL
LIN {X 0,Y 509.833,Z 194.289,A -85,B 0,C 180,E1 -5440.383,E2 -5440.383} C_VEL
LIN {X 0,Y 509.818,Z 194.298,A -85,B 0,C 180,E1 -5443.063,E2 -5443.063} C_VEL
LIN {X 0,Y 509.825,Z 194.292,A -85,B 0,C 180,E1 -5445.793,E2 -5445.793} C_VEL
LIN {X 0,Y 509.85,Z 194.29,A -85,B 0,C 180,E1 -5448.575,E2 -5448.575} C_VEL
LIN {X 0,Y 509.846,Z 194.287,A -85,B 0,C 180,E1 -5451.787,E2 -5451.787} C_VEL
LIN {X 0,Y 509.825,Z 194.294,A -85,B 0,C 180,E1 -5454.622,E2 -5454.622} C_VEL
LIN {X 0,Y 509.857,Z 194.287,A -85,B 0,C 180,E1 -5457.481,E2 -5457.481} C_VEL
LIN {X 0,Y 509.89,Z 194.481,A -85,B 0,C 180,E1 -5459.163,E2 -5459.163} C_VEL
LIN {X 0,Y 515.443,Z 213.013,A -85,B 0,C 180,E1 -5461.391,E2 -5461.391} C_VEL
LIN {X 0,Y 515.542,Z 217.407,A -85,B 0,C 180,E1 -5461.835,E2 -5461.835} C_VEL
LIN {X 0,Y 514.893,Z 233.333,A -85,B 0,C 180,E1 -5463.37,E2 -5463.37} C_VEL
LIN {X 0,Y 518.074,Z 251.415,A -85,B 0,C 180,E1 -5463.822,E2 -5463.822} C_VEL
LIN {X 0,Y 516.203,Z 439.773,A -85,B 0,C 180,E1 -5466.586,E2 -5466.586} C_VEL
LIN {X 0,Y 515.845,Z 455.04,A -85,B 0,C 180,E1 -5466.94,E2 -5466.94} C_VEL
LIN {X 0,Y 515.335,Z 470.782,A -85,B 0,C 180,E1 -5467.446,E2 -5467.446} C_VEL
LIN {X 0,Y 514.739,Z 485.229,A -85,B 0,C 180,E1 -5468.049,E2 -5468.049} C_VEL
LIN {X 0,Y 514.075,Z 500.743,A -85,B 0,C 180,E1 -5468.865,E2 -5468.865} C_VEL
LIN {X 0,Y 513.339,Z 515.039,A -85,B 0,C 180,E1 -5469.777,E2 -5469.777} C_VEL
LIN {X 0,Y 512.637,Z 528.455,A -85,B 0,C 180,E1 -5470.791,E2 -5470.791} C_VEL
LIN {X 0,Y 511.906,Z 542.004,A -85,B 0,C 180,E1 -5472.007,E2 -5472.007} C_VEL
LIN {X 0,Y 511.291,Z 553.52,A -85,B 0,C 180,E1 -5473.223,E2 -5473.223} C_VEL
LIN {X 0,Y 510.715,Z 565.499,A -85,B 0,C 180,E1 -5474.696,E2 -5474.696} C_VEL
LIN {X 0,Y 510.238,Z 574.995,A -85,B 0,C 180,E1 -5476.052,E2 -5476.052} C_VEL
LIN {X 0,Y 509.901,Z 584.528,A -85,B 0,C 180,E1 -5477.665,E2 -5477.665} C_VEL
LIN {X 0,Y 509.621,Z 592.505,A -85,B 0,C 180,E1 -5479.271,E2 -5479.271} C_VEL
LIN {X 0,Y 509.393,Z 599.161,A -85,B 0,C 180,E1 -5480.871,E2 -5480.871} C_VEL
LIN {X 0,Y 509.3,Z 604.559,A -85,B 0,C 180,E1 -5482.468,E2 -5482.468} C_VEL
LIN {X 0,Y 509.255,Z 607.895,A -85,B 0,C 180,E1 -5483.662,E2 -5483.662} C_VEL
LIN {X 0,Y 509.142,Z 611.318,A -85,B 0,C 180,E1 -5485.25,E2 -5485.25} C_VEL
LIN {X 0,Y 509.183,Z 613.81,A -85,B 0,C 180,E1 -5486.835,E2 -5486.835} C_VEL
LIN {X 0,Y 509.107,Z 615.212,A -85,B 0,C 180,E1 -5488.418,E2 -5488.418} C_VEL
LIN {X 0,Y 509.061,Z 615.741,A -85,B 0,C 180,E1 -5490,E2 -5490} C_VEL
LIN {X 0,Y 509.107,Z 615.214,A -85,B 0,C 180,E1 -5491.582,E2 -5491.582} C_VEL
LIN {X 0,Y 509.183,Z 613.813,A -85,B 0,C 180,E1 -5493.165,E2 -5493.165} C_VEL
LIN {X 0,Y 509.142,Z 611.325,A -85,B 0,C 180,E1 -5494.751,E2 -5494.751} C_VEL
LIN {X 0,Y 509.26,Z 607.546,A -85,B 0,C 180,E1 -5496.473,E2 -5496.473} C_VEL
LIN {X 0,Y 509.353,Z 602.057,A -85,B 0,C 180,E1 -5498.33,E2 -5498.33} C_VEL
LIN {X 0,Y 509.536,Z 594.36,A -85,B 0,C 180,E1 -5500.33,E2 -5500.33} C_VEL
LIN {X 0,Y 509.868,Z 585.674,A -85,B 0,C 180,E1 -5502.134,E2 -5502.134} C_VEL
LIN {X 0,Y 510.207,Z 576.295,A -85,B 0,C 180,E1 -5503.746,E2 -5503.746} C_VEL
LIN {X 0,Y 510.661,Z 566.644,A -85,B 0,C 180,E1 -5505.158,E2 -5505.158} C_VEL
LIN {X 0,Y 511.198,Z 555.395,A -85,B 0,C 180,E1 -5506.575,E2 -5506.575} C_VEL
LIN {X 0,Y 511.847,Z 543.146,A -85,B 0,C 180,E1 -5507.892,E2 -5507.892} C_VEL
LIN {X 0,Y 512.613,Z 529.586,A -85,B 0,C 180,E1 -5509.121,E2 -5509.121} C_VEL
LIN {X 0,Y 513.299,Z 516.609,A -85,B 0,C 180,E1 -5510.121,E2 -5510.121} C_VEL
LIN {X 0,Y 513.95,Z 502.667,A -85,B 0,C 180,E1 -5511.036,E2 -5511.036} C_VEL
LIN {X 0,Y 514.711,Z 488.032,A -85,B 0,C 180,E1 -5511.823,E2 -5511.823} C_VEL
LIN {X 0,Y 515.302,Z 472.298,A -85,B 0,C 180,E1 -5512.503,E2 -5512.503} C_VEL
LIN {X 0,Y 515.829,Z 456.21,A -85,B 0,C 180,E1 -5513.034,E2 -5513.034} C_VEL
LIN {X 0,Y 516.223,Z 440.088,A -85,B 0,C 180,E1 -5513.414,E2 -5513.414} C_VEL
LIN {X 0,Y 518.06,Z 255.497,A -85,B 0,C 180,E1 -5516.121,E2 -5516.121} C_VEL
LIN {X 0,Y 517.968,Z 250.162,A -85,B 0,C 180,E1 -5516.207,E2 -5516.207} C_VEL
LIN {X 0,Y 514.96,Z 233.246,A -85,B 0,C 180,E1 -5516.656,E2 -5516.656} C_VEL
LIN {X 0,Y 515.742,Z 214.359,A -85,B 0,C 180,E1 -5518.486,E2 -5518.486} C_VEL
LIN {X 0,Y 511.331,Z 199.376,A -85,B 0,C 180,E1 -5520.267,E2 -5520.267} C_VEL
LIN {X 0,Y 509.868,Z 194.287,A -85,B 0,C 180,E1 -5520.914,E2 -5520.914} C_VEL
LIN {X 0,Y 509.856,Z 194.281,A -85,B 0,C 180,E1 -5523.461,E2 -5523.461} C_VEL
LIN {X 0,Y 509.807,Z 194.293,A -85,B 0,C 180,E1 -5526.354,E2 -5526.354} C_VEL
LIN {X 0,Y 509.843,Z 194.289,A -85,B 0,C 180,E1 -5529.352,E2 -5529.352} C_VEL
LIN {X 0,Y 509.812,Z 194.291,A -85,B 0,C 180,E1 -5532.492,E2 -5532.492} C_VEL
LIN {X 0,Y 509.836,Z 194.287,A -85,B 0,C 180,E1 -5535.33,E2 -5535.33} C_VEL
LIN {X 0,Y 509.849,Z 194.289,A -85,B 0,C 180,E1 -5538.574,E2 -5538.574} C_VEL
LIN {X 0,Y 509.846,Z 194.286,A -85,B 0,C 180,E1 -5541.787,E2 -5541.787} C_VEL
LIN {X 0,Y 509.826,Z 194.287,A -85,B 0,C 180,E1 -5544.622,E2 -5544.622} C_VEL
LIN {X 0,Y 509.856,Z 194.28,A -85,B 0,C 180,E1 -5547.481,E2 -5547.481} C_VEL
LIN {X 0,Y 509.855,Z 194.284,A -85,B 0,C 180,E1 -5550.274,E2 -5550.274} C_VEL
LIN {X 0,Y 509.879,Z 194.279,A -85,B 0,C 180,E1 -5552.944,E2 -5552.944} C_VEL
LIN {X 0,Y 509.846,Z 194.283,A -85,B 0,C 180,E1 -5555.573,E2 -5555.573} C_VEL
LIN {X 0,Y 509.818,Z 194.291,A -85,B 0,C 180,E1 -5558.149,E2 -5558.149} C_VEL
LIN {X 0,Y 509.854,Z 194.28,A -85,B 0,C 180,E1 -5560.681,E2 -5560.681} C_VEL
LIN {X 0,Y 509.864,Z 194.283,A -85,B 0,C 180,E1 -5563.174,E2 -5563.174} C_VEL
LIN {X 0,Y 509.859,Z 194.282,A -85,B 0,C 180,E1 -5565.634,E2 -5565.634} C_VEL
LIN {X 0,Y 509.909,Z 194.272,A -85,B 0,C 180,E1 -5568.874,E2 -5568.874} C_VEL
LIN {X 0,Y 509.918,Z 194.279,A -85,B 0,C 180,E1 -5572.078,E2 -5572.078} C_VEL
LIN {X 0,Y 509.973,Z 194.27,A -85,B 0,C 180,E1 -5574.464,E2 -5574.464} C_VEL
LIN {X 0,Y 510.048,Z 194.245,A -85,B 0,C 180,E1 -5577.631,E2 -5577.631} C_VEL
LIN {X 0,Y 510.061,Z 194.26,A -85,B 0,C 180,E1 -5580.789,E2 -5580.789} C_VEL
LIN {X 0,Y 509.95,Z 194.27,A -85,B 0,C 180,E1 -5583.16,E2 -5583.16} C_VEL
LIN {X 0,Y 509.974,Z 194.273,A -85,B 0,C 180,E1 -5586.33,E2 -5586.33} C_VEL
LIN {X 0,Y 509.908,Z 194.278,A -85,B 0,C 180,E1 -5588.72,E2 -5588.72} C_VEL
LIN {X 0,Y 509.901,Z 194.277,A -85,B 0,C 180,E1 -5591.932,E2 -5591.932} C_VEL
LIN {X 0,Y 509.891,Z 194.279,A -85,B 0,C 180,E1 -5595.242,E2 -5595.242} C_VEL
LIN {X 0,Y 509.886,Z 194.279,A -85,B 0,C 180,E1 -5598.001,E2 -5598.001} C_VEL
LIN {X 0,Y 509.847,Z 194.283,A -85,B 0,C 180,E1 -5601.002,E2 -5601.002} C_VEL
LIN {X 0,Y 509.867,Z 194.278,A -85,B 0,C 180,E1 -5604.426,E2 -5604.426} C_VEL
LIN {X 0,Y 509.883,Z 194.277,A -85,B 0,C 180,E1 -5607.056,E2 -5607.056} C_VEL
LIN {X 0,Y 509.878,Z 194.287,A -85,B 0,C 180,E1 -5609.75,E2 -5609.75} C_VEL
LIN {X 0,Y 509.872,Z 194.276,A -85,B 0,C 180,E1 -5612.774,E2 -5612.774} C_VEL
LIN {X 0,Y 509.84,Z 194.293,A -85,B 0,C 180,E1 -5615.581,E2 -5615.581} C_VEL
LIN {X 0,Y 509.847,Z 194.28,A -85,B 0,C 180,E1 -5618.338,E2 -5618.338} C_VEL
LIN {X 0,Y 509.855,Z 194.29,A -85,B 0,C 180,E1 -5621.425,E2 -5621.425} C_VEL
LIN {X 0,Y 509.836,Z 194.282,A -85,B 0,C 180,E1 -5624.67,E2 -5624.67} C_VEL
LIN {X 0,Y 509.831,Z 194.292,A -85,B 0,C 180,E1 -5627.51,E2 -5627.51} C_VEL
LIN {X 0,Y 509.844,Z 194.284,A -85,B 0,C 180,E1 -5630.648,E2 -5630.648} C_VEL
LIN {X 0,Y 509.819,Z 194.287,A -85,B 0,C 180,E1 -5633.74,E2 -5633.74} C_VEL
LIN {X 0,Y 509.152,Z 194.369,A -85,B 0,C 180,E1 -5634.4,E2 -5634.4} C_VEL
LIN {X 0,Y 506.339,Z 194.729,A -85,B 0,C 180,E1 -5635.472,E2 -5635.472} C_VEL
LIN {X 0,Y 503.951,Z 195.028,A -85,B 0,C 180,E1 -5636.336,E2 -5636.336} C_VEL
LIN {X 0,Y 502.904,Z 195.154,A -85,B 0,C 180,E1 -5637.002,E2 -5637.002} C_VEL
LIN {X 0,Y 502.807,Z 195.163,A -85,B 0,C 180,E1 -5637.228,E2 -5637.228} C_VEL
LIN {X 0,Y 502.814,Z 195.162,A -85,B 0,C 180,E1 -5640.065,E2 -5640.065} C_VEL
LIN {X 0,Y 502.831,Z 195.157,A -85,B 0,C 180,E1 -5642.533,E2 -5642.533} C_VEL
LIN {X 0,Y 502.826,Z 195.163,A -85,B 0,C 180,E1 -5645.299,E2 -5645.299} C_VEL
LIN {X 0,Y 502.779,Z 195.167,A -85,B 0,C 180,E1 -5647.826,E2 -5647.826} C_VEL
LIN {X 0,Y 502.823,Z 195.154,A -85,B 0,C 180,E1 -5650.4,E2 -5650.4} C_VEL
LIN {X 0,Y 502.819,Z 195.164,A -85,B 0,C 180,E1 -5652.931,E2 -5652.931} C_VEL
LIN {X 0,Y 502.844,Z 195.151,A -85,B 0,C 180,E1 -5655.429,E2 -5655.429} C_VEL
LIN {X 0,Y 502.877,Z 195.16,A -85,B 0,C 180,E1 -5658.717,E2 -5658.717} C_VEL
LIN {X 0,Y 502.901,Z 195.153,A -85,B 0,C 180,E1 -5661.967,E2 -5661.967} C_VEL
LIN {X 0,Y 502.93,Z 195.147,A -85,B 0,C 180,E1 -5664.386,E2 -5664.386} C_VEL
LIN {X 0,Y 502.972,Z 195.265,A -85,B 0,C 180,E1 -5667.297,E2 -5667.297} C_VEL
LIN {X 0,Y 506.644,Z 207.999,A -85,B 0,C 180,E1 -5668.966,E2 -5668.966} C_VEL
LIN {X 0,Y 510.328,Z 216.633,A -85,B 0,C 180,E1 -5669.314,E2 -5669.314} C_VEL
LIN {X 0,Y 511.845,Z 224.393,A -85,B 0,C 180,E1 -5669.52,E2 -5669.52} C_VEL
LIN {X 0,Y 509.808,Z 413.943,A -85,B 0,C 180,E1 -5672.345,E2 -5672.345} C_VEL
LIN {X 0,Y 509.422,Z 430.821,A -85,B 0,C 180,E1 -5672.767,E2 -5672.767} C_VEL
LIN {X 0,Y 508.801,Z 446.598,A -85,B 0,C 180,E1 -5673.316,E2 -5673.316} C_VEL
LIN {X 0,Y 508.14,Z 462.601,A -85,B 0,C 180,E1 -5674.044,E2 -5674.044} C_VEL
LIN {X 0,Y 507.426,Z 477.163,A -85,B 0,C 180,E1 -5674.866,E2 -5674.866} C_VEL
LIN {X 0,Y 506.625,Z 491.799,A -85,B 0,C 180,E1 -5675.872,E2 -5675.872} C_VEL
LIN {X 0,Y 505.847,Z 505.262,A -85,B 0,C 180,E1 -5676.982,E2 -5676.982} C_VEL
LIN {X 0,Y 505.07,Z 518.522,A -85,B 0,C 180,E1 -5678.275,E2 -5678.275} C_VEL
LIN {X 0,Y 504.321,Z 530.322,A -85,B 0,C 180,E1 -5679.626,E2 -5679.626} C_VEL
LIN {X 0,Y 503.722,Z 541.025,A -85,B 0,C 180,E1 -5681.06,E2 -5681.06} C_VEL
LIN {X 0,Y 503.214,Z 551.249,A -85,B 0,C 180,E1 -5682.686,E2 -5682.686} C_VEL
LIN {X 0,Y 502.777,Z 560.108,A -85,B 0,C 180,E1 -5684.366,E2 -5684.366} C_VEL
LIN {X 0,Y 502.487,Z 566.612,A -85,B 0,C 180,E1 -5685.827,E2 -5685.827} C_VEL
LIN {X 0,Y 502.332,Z 572.802,A -85,B 0,C 180,E1 -5687.505,E2 -5687.505} C_VEL
LIN {X 0,Y 502.18,Z 577.781,A -85,B 0,C 180,E1 -5689.2,E2 -5689.2} C_VEL
LIN {X 0,Y 502.084,Z 580.791,A -85,B 0,C 180,E1 -5690.483,E2 -5690.483} C_VEL
LIN {X 0,Y 501.986,Z 584.168,A -85,B 0,C 180,E1 -5692.479,E2 -5692.479} C_VEL
LIN {X 0,Y 501.94,Z 586.054,A -85,B 0,C 180,E1 -5694.48,E2 -5694.48} C_VEL
LIN {X 0,Y 501.983,Z 586.493,A -85,B 0,C 180,E1 -5696.359,E2 -5696.359} C_VEL
LIN {X 0,Y 501.99,Z 585.485,A -85,B 0,C 180,E1 -5698.424,E2 -5698.424} C_VEL
LIN {X 0,Y 502.039,Z 583.284,A -85,B 0,C 180,E1 -5700.262,E2 -5700.262} C_VEL
LIN {X 0,Y 502.162,Z 579.667,A -85,B 0,C 180,E1 -5702.128,E2 -5702.128} C_VEL
LIN {X 0,Y 502.273,Z 574.564,A -85,B 0,C 180,E1 -5704.034,E2 -5704.034} C_VEL
LIN {X 0,Y 502.439,Z 568.554,A -85,B 0,C 180,E1 -5705.778,E2 -5705.778} C_VEL
LIN {X 0,Y 502.715,Z 561.154,A -85,B 0,C 180,E1 -5707.52,E2 -5707.52} C_VEL
LIN {X 0,Y 503.096,Z 552.643,A -85,B 0,C 180,E1 -5709.172,E2 -5709.172} C_VEL
LIN {X 0,Y 503.619,Z 543.127,A -85,B 0,C 180,E1 -5710.721,E2 -5710.721} C_VEL
LIN {X 0,Y 504.189,Z 532.522,A -85,B 0,C 180,E1 -5712.196,E2 -5712.196} C_VEL
LIN {X 0,Y 504.969,Z 520.285,A -85,B 0,C 180,E1 -5713.638,E2 -5713.638} C_VEL
LIN {X 0,Y 505.71,Z 508.064,A -85,B 0,C 180,E1 -5714.866,E2 -5714.866} C_VEL
LIN {X 0,Y 506.495,Z 493.841,A -85,B 0,C 180,E1 -5716.069,E2 -5716.069} C_VEL
LIN {X 0,Y 507.331,Z 479.282,A -85,B 0,C 180,E1 -5717.093,E2 -5717.093} C_VEL
LIN {X 0,Y 508.092,Z 463.656,A -85,B 0,C 180,E1 -5717.998,E2 -5717.998} C_VEL
LIN {X 0,Y 508.79,Z 448.227,A -85,B 0,C 180,E1 -5718.712,E2 -5718.712} C_VEL
LIN {X 0,Y 509.343,Z 432.636,A -85,B 0,C 180,E1 -5719.275,E2 -5719.275} C_VEL
LIN {X 0,Y 509.796,Z 415.947,A -85,B 0,C 180,E1 -5719.701,E2 -5719.701} C_VEL
LIN {X 0,Y 510.114,Z 387.012,A -85,B 0,C 180,E1 -5720.164,E2 -5720.164} C_VEL
LIN {X 0,Y 511.83,Z 223.994,A -85,B 0,C 180,E1 -5722.585,E2 -5722.585} C_VEL
LIN {X 0,Y 510.1,Z 216.088,A -85,B 0,C 180,E1 -5722.808,E2 -5722.808} C_VEL
LIN {X 0,Y 506.425,Z 207.812,A -85,B 0,C 180,E1 -5723.177,E2 -5723.177} C_VEL
LIN {X 0,Y 502.781,Z 195.17,A -85,B 0,C 180,E1 -5724.911,E2 -5724.911} C_VEL
LIN {X 0,Y 502.774,Z 195.171,A -85,B 0,C 180,E1 -5727.915,E2 -5727.915} C_VEL
LIN {X 0,Y 502.804,Z 195.168,A -85,B 0,C 180,E1 -5730.711,E2 -5730.711} C_VEL
LIN {X 0,Y 502.767,Z 195.171,A -85,B 0,C 180,E1 -5733.459,E2 -5733.459} C_VEL
LIN {X 0,Y 502.759,Z 195.169,A -85,B 0,C 180,E1 -5736.085,E2 -5736.085} C_VEL
LIN {X 0,Y 502.773,Z 195.169,A -85,B 0,C 180,E1 -5738.688,E2 -5738.688} C_VEL
LIN {X 0,Y 502.818,Z 195.164,A -85,B 0,C 180,E1 -5741.248,E2 -5741.248} C_VEL
LIN {X 0,Y 502.841,Z 195.159,A -85,B 0,C 180,E1 -5744.6,E2 -5744.6} C_VEL
LIN {X 0,Y 502.869,Z 195.152,A -85,B 0,C 180,E1 -5748.039,E2 -5748.039} C_VEL
LIN {X 0,Y 502.859,Z 195.156,A -85,B 0,C 180,E1 -5751.156,E2 -5751.156} C_VEL
LIN {X 0,Y 502.898,Z 195.149,A -85,B 0,C 180,E1 -5753.581,E2 -5753.581} C_VEL
LIN {X 0,Y 502.891,Z 195.155,A -85,B 0,C 180,E1 -5756.795,E2 -5756.795} C_VEL
LIN {X 0,Y 503.027,Z 195.135,A -85,B 0,C 180,E1 -5759.199,E2 -5759.199} C_VEL
LIN {X 0,Y 502.892,Z 195.152,A -85,B 0,C 180,E1 -5761.602,E2 -5761.602} C_VEL
LIN {X 0,Y 502.891,Z 195.149,A -85,B 0,C 180,E1 -5763.205,E2 -5763.205} C_VEL
LIN {X 0,Y 502.92,Z 195.153,A -85,B 0,C 180,E1 -5766.419,E2 -5766.419} C_VEL
LIN {X 0,Y 502.868,Z 195.154,A -85,B 0,C 180,E1 -5768.843,E2 -5768.843} C_VEL
LIN {X 0,Y 502.839,Z 195.165,A -85,B 0,C 180,E1 -5772.102,E2 -5772.102} C_VEL
LIN {X 0,Y 502.842,Z 195.16,A -85,B 0,C 180,E1 -5775.4,E2 -5775.4} C_VEL
LIN {X 0,Y 502.84,Z 195.161,A -85,B 0,C 180,E1 -5778.123,E2 -5778.123} C_VEL
LIN {X 0,Y 502.822,Z 195.161,A -85,B 0,C 180,E1 -5780.536,E2 -5780.536} C_VEL
LIN {X 0,Y 502.79,Z 195.165,A -85,B 0,C 180,E1 -5783.041,E2 -5783.041} C_VEL
LIN {X 0,Y 502.836,Z 195.165,A -85,B 0,C 180,E1 -5785.676,E2 -5785.676} C_VEL
LIN {X 0,Y 502.834,Z 195.159,A -85,B 0,C 180,E1 -5788.373,E2 -5788.373} C_VEL
LIN {X 0,Y 502.791,Z 195.17,A -85,B 0,C 180,E1 -5791.5,E2 -5791.5} C_VEL
LIN {X 0,Y 502.798,Z 195.165,A -85,B 0,C 180,E1 -5794.445,E2 -5794.445} C_VEL
LIN {X 0,Y 502.772,Z 195.175,A -85,B 0,C 180,E1 -5797.178,E2 -5797.178} C_VEL
LIN {X 0,Y 502.783,Z 195.168,A -85,B 0,C 180,E1 -5800.015,E2 -5800.015} C_VEL
LIN {X 0,Y 502.797,Z 195.166,A -85,B 0,C 180,E1 -5802.2,E2 -5802.2} C_VEL
LIN {X 0,Y 502.795,Z 195.17,A -85,B 0,C 180,E1 -5805.469,E2 -5805.469} C_VEL
LIN {X 0,Y 502.815,Z 195.168,A -85,B 0,C 180,E1 -5808.935,E2 -5808.935} C_VEL
LIN {X 0,Y 502.788,Z 195.166,A -85,B 0,C 180,E1 -5812.047,E2 -5812.047} C_VEL
LIN {X 0,Y 502.794,Z 195.17,A -85,B 0,C 180,E1 -5815.035,E2 -5815.035} C_VEL
LIN {X 0,Y 502.779,Z 195.168,A -85,B 0,C 180,E1 -5817.916,E2 -5817.916} C_VEL
LIN {X 0,Y 502.803,Z 195.169,A -85,B 0,C 180,E1 -5818.769,E2 -5818.769} C_VEL
LIN {X 0,Y 508.754,Z 214.982,A -85,B 0,C 180,E1 -5821.2,E2 -5821.2} C_VEL
LIN {X 0,Y 508.996,Z 217.206,A -85,B 0,C 180,E1 -5821.44,E2 -5821.44} C_VEL
LIN {X 0,Y 508.263,Z 232.935,A -85,B 0,C 180,E1 -5822.983,E2 -5822.983} C_VEL
LIN {X 0,Y 511.669,Z 251.82,A -85,B 0,C 180,E1 -5823.477,E2 -5823.477} C_VEL
LIN {X 0,Y 509.728,Z 437.862,A -85,B 0,C 180,E1 -5826.243,E2 -5826.243} C_VEL
LIN {X 0,Y 509.26,Z 454.696,A -85,B 0,C 180,E1 -5826.625,E2 -5826.625} C_VEL
LIN {X 0,Y 508.753,Z 470.47,A -85,B 0,C 180,E1 -5827.138,E2 -5827.138} C_VEL
LIN {X 0,Y 508.055,Z 486.14,A -85,B 0,C 180,E1 -5827.802,E2 -5827.802} C_VEL
LIN {X 0,Y 507.29,Z 502.44,A -85,B 0,C 180,E1 -5828.687,E2 -5828.687} C_VEL
LIN {X 0,Y 506.511,Z 516.203,A -85,B 0,C 180,E1 -5829.598,E2 -5829.598} C_VEL
LIN {X 0,Y 505.753,Z 529.457,A -85,B 0,C 180,E1 -5830.632,E2 -5830.632} C_VEL
LIN {X 0,Y 504.988,Z 542.798,A -85,B 0,C 180,E1 -5831.857,E2 -5831.857} C_VEL
LIN {X 0,Y 504.274,Z 555.07,A -85,B 0,C 180,E1 -5833.191,E2 -5833.191} C_VEL
LIN {X 0,Y 503.692,Z 566.339,A -85,B 0,C 180,E1 -5834.627,E2 -5834.627} C_VEL
LIN {X 0,Y 503.148,Z 577.253,A -85,B 0,C 180,E1 -5836.264,E2 -5836.264} C_VEL
LIN {X 0,Y 502.788,Z 586.428,A -85,B 0,C 180,E1 -5837.897,E2 -5837.897} C_VEL
LIN {X 0,Y 502.489,Z 594.109,A -85,B 0,C 180,E1 -5839.524,E2 -5839.524} C_VEL
LIN {X 0,Y 502.256,Z 601.818,A -85,B 0,C 180,E1 -5841.552,E2 -5841.552} C_VEL
LIN {X 0,Y 502.183,Z 607.682,A -85,B 0,C 180,E1 -5843.572,E2 -5843.572} C_VEL
LIN {X 0,Y 502.061,Z 611.107,A -85,B 0,C 180,E1 -5845.182,E2 -5845.182} C_VEL
LIN {X 0,Y 502.101,Z 613.602,A -85,B 0,C 180,E1 -5846.791,E2 -5846.791} C_VEL
LIN {X 0,Y 502.031,Z 615.006,A -85,B 0,C 180,E1 -5848.396,E2 -5848.396} C_VEL
LIN {X 0,Y 501.975,Z 615.537,A -85,B 0,C 180,E1 -5850,E2 -5850} C_VEL
LIN {X 0,Y 502.031,Z 615.01,A -85,B 0,C 180,E1 -5851.605,E2 -5851.605} C_VEL
LIN {X 0,Y 502.101,Z 613.609,A -85,B 0,C 180,E1 -5853.21,E2 -5853.21} C_VEL
LIN {X 0,Y 502.061,Z 611.121,A -85,B 0,C 180,E1 -5854.818,E2 -5854.818} C_VEL
LIN {X 0,Y 502.183,Z 607.595,A -85,B 0,C 180,E1 -5856.469,E2 -5856.469} C_VEL
LIN {X 0,Y 502.257,Z 601.848,A -85,B 0,C 180,E1 -5858.449,E2 -5858.449} C_VEL
LIN {X 0,Y 502.49,Z 594.148,A -85,B 0,C 180,E1 -5860.476,E2 -5860.476} C_VEL
LIN {X 0,Y 502.839,Z 585.46,A -85,B 0,C 180,E1 -5862.307,E2 -5862.307} C_VEL
LIN {X 0,Y 503.201,Z 576.077,A -85,B 0,C 180,E1 -5863.941,E2 -5863.941} C_VEL
LIN {X 0,Y 503.697,Z 566.422,A -85,B 0,C 180,E1 -5865.373,E2 -5865.373} C_VEL
LIN {X 0,Y 504.278,Z 555.168,A -85,B 0,C 180,E1 -5866.809,E2 -5866.809} C_VEL
LIN {X 0,Y 504.98,Z 542.915,A -85,B 0,C 180,E1 -5868.144,E2 -5868.144} C_VEL
LIN {X 0,Y 505.778,Z 529.585,A -85,B 0,C 180,E1 -5869.369,E2 -5869.369} C_VEL
LIN {X 0,Y 506.553,Z 516.365,A -85,B 0,C 180,E1 -5870.401,E2 -5870.401} C_VEL
LIN {X 0,Y 507.256,Z 502.617,A -85,B 0,C 180,E1 -5871.315,E2 -5871.315} C_VEL
LIN {X 0,Y 508.073,Z 487.771,A -85,B 0,C 180,E1 -5872.123,E2 -5872.123} C_VEL
LIN {X 0,Y 508.669,Z 473.323,A -85,B 0,C 180,E1 -5872.759,E2 -5872.759} C_VEL
LIN {X 0,Y 509.256,Z 456.82,A -85,B 0,C 180,E1 -5873.322,E2 -5873.322} C_VEL
LIN {X 0,Y 509.682,Z 441.189,A -85,B 0,C 180,E1 -5873.705,E2 -5873.705} C_VEL
LIN {X 0,Y 510.641,Z 348.386,A -85,B 0,C 180,E1 -5875.093,E2 -5875.093} C_VEL
LIN {X 0,Y 511.592,Z 251.312,A -85,B 0,C 180,E1 -5876.537,E2 -5876.537} C_VEL
LIN {X 0,Y 508.332,Z 233.251,A -85,B 0,C 180,E1 -5877.011,E2 -5877.011} C_VEL
LIN {X 0,Y 509.095,Z 216.385,A -85,B 0,C 180,E1 -5878.667,E2 -5878.667} C_VEL
LIN {X 0,Y 503.927,Z 198.785,A -85,B 0,C 180,E1 -5880.796,E2 -5880.796} C_VEL
LIN {X 0,Y 502.813,Z 195.169,A -85,B 0,C 180,E1 -5881.275,E2 -5881.275} C_VEL
LIN {X 0,Y 502.801,Z 195.166,A -85,B 0,C 180,E1 -5883.994,E2 -5883.994} C_VEL
LIN {X 0,Y 502.762,Z 195.173,A -85,B 0,C 180,E1 -5887.176,E2 -5887.176} C_VEL
LIN {X 0,Y 502.783,Z 195.163,A -85,B 0,C 180,E1 -5890.015,E2 -5890.015} C_VEL
LIN {X 0,Y 502.801,Z 195.163,A -85,B 0,C 180,E1 -5892.199,E2 -5892.199} C_VEL
LIN {X 0,Y 502.782,Z 195.164,A -85,B 0,C 180,E1 -5895.47,E2 -5895.47} C_VEL
LIN {X 0,Y 502.792,Z 195.165,A -85,B 0,C 180,E1 -5897.86,E2 -5897.86} C_VEL
LIN {X 0,Y 502.793,Z 195.172,A -85,B 0,C 180,E1 -5901.023,E2 -5901.023} C_VEL
LIN {X 0,Y 502.771,Z 195.161,A -85,B 0,C 180,E1 -5904.169,E2 -5904.169} C_VEL
LIN {X 0,Y 502.827,Z 195.161,A -85,B 0,C 180,E1 -5906.994,E2 -5906.994} C_VEL
LIN {X 0,Y 502.811,Z 195.16,A -85,B 0,C 180,E1 -5910.065,E2 -5910.065} C_VEL
LIN {X 0,Y 502.825,Z 195.165,A -85,B 0,C 180,E1 -5912.533,E2 -5912.533} C_VEL
LIN {X 0,Y 502.783,Z 195.164,A -85,B 0,C 180,E1 -5915.309,E2 -5915.309} C_VEL
LIN {X 0,Y 502.776,Z 195.166,A -85,B 0,C 180,E1 -5917.826,E2 -5917.826} C_VEL
LIN {X 0,Y 502.816,Z 195.157,A -85,B 0,C 180,E1 -5920.4,E2 -5920.4} C_VEL
LIN {X 0,Y 502.81,Z 195.164,A -85,B 0,C 180,E1 -5922.931,E2 -5922.931} C_VEL
LIN {X 0,Y 502.84,Z 195.156,A -85,B 0,C 180,E1 -5925.429,E2 -5925.429} C_VEL
LIN {X 0,Y 502.873,Z 195.147,A -85,B 0,C 180,E1 -5928.717,E2 -5928.717} C_VEL
LIN {X 0,Y 502.877,Z 195.154,A -85,B 0,C 180,E1 -5931.966,E2 -5931.966} C_VEL
LIN {X 0,Y 502.927,Z 195.148,A -85,B 0,C 180,E1 -5934.386,E2 -5934.386} C_VEL
LIN {X 0,Y 503.018,Z 195.12,A -85,B 0,C 180,E1 -5937.598,E2 -5937.598} C_VEL
LIN {X 0,Y 503.022,Z 195.135,A -85,B 0,C 180,E1 -5940,E2 -5940} C_VEL
LIN {X 0,Y 503.019,Z 195.139,A -85,B 0,C 180,E1 -5942.402,E2 -5942.402} C_VEL
LIN {X 0,Y 502.933,Z 195.138,A -85,B 0,C 180,E1 -5945.614,E2 -5945.614} C_VEL
LIN {X 0,Y 502.897,Z 195.156,A -85,B 0,C 180,E1 -5948.033,E2 -5948.033} C_VEL
LIN {X 0,Y 502.874,Z 195.148,A -85,B 0,C 180,E1 -5951.283,E2 -5951.283} C_VEL
LIN {X 0,Y 502.842,Z 195.158,A -85,B 0,C 180,E1 -5954.571,E2 -5954.571} C_VEL
LIN {X 0,Y 502.859,Z 195.155,A -85,B 0,C 180,E1 -5957.907,E2 -5957.907} C_VEL
LIN {X 0,Y 502.826,Z 195.159,A -85,B 0,C 180,E1 -5960.536,E2 -5960.536} C_VEL
LIN {X 0,Y 502.791,Z 195.163,A -85,B 0,C 180,E1 -5963.04,E2 -5963.04} C_VEL
LIN {X 0,Y 502.838,Z 195.156,A -85,B 0,C 180,E1 -5965.676,E2 -5965.676} C_VEL
LIN {X 0,Y 502.839,Z 195.159,A -85,B 0,C 180,E1 -5968.373,E2 -5968.373} C_VEL
LIN {X 0,Y 502.792,Z 195.165,A -85,B 0,C 180,E1 -5971.499,E2 -5971.499} C_VEL
LIN {X 0,Y 502.804,Z 195.162,A -85,B 0,C 180,E1 -5974.445,E2 -5974.445} C_VEL
LIN {X 0,Y 502.778,Z 195.166,A -85,B 0,C 180,E1 -5977.178,E2 -5977.178} C_VEL
LIN {X 0,Y 502.785,Z 195.167,A -85,B 0,C 180,E1 -5980.015,E2 -5980.015} C_VEL
LIN {X 0,Y 502.8,Z 195.162,A -85,B 0,C 180,E1 -5982.199,E2 -5982.199} C_VEL
LIN {X 0,Y 502.784,Z 195.169,A -85,B 0,C 180,E1 -5985.47,E2 -5985.47} C_VEL
LIN {X 0,Y 502.817,Z 195.159,A -85,B 0,C 180,E1 -5988.934,E2 -5988.934} C_VEL
LIN {X 0,Y 502.791,Z 195.164,A -85,B 0,C 180,E1 -5992.046,E2 -5992.046} C_VEL
LIN {X 0,Y 502.799,Z 195.162,A -85,B 0,C 180,E1 -5995.034,E2 -5995.034} C_VEL
LIN {X 0,Y 502.807,Z 195.163,A -85,B 0,C 180,E1 -5997.228,E2 -5997.228} C_VEL
LIN {X 0,Y 502.106,Z 195.247,A -85,B 0,C 180,E1 -5997.896,E2 -5997.896} C_VEL
LIN {X 0,Y 499.241,Z 195.606,A -85,B 0,C 180,E1 -5998.982,E2 -5998.982} C_VEL
LIN {X 0,Y 496.846,Z 195.906,A -85,B 0,C 180,E1 -5999.857,E2 -5999.857} C_VEL
LIN {X 0,Y 495.83,Z 196.032,A -85,B 0,C 180,E1 -6000.533,E2 -6000.533} C_VEL
LIN {X 0,Y 495.752,Z 196.043,A -85,B 0,C 180,E1 -6000.761,E2 -6000.761} C_VEL
LIN {X 0,Y 495.79,Z 196.037,A -85,B 0,C 180,E1 -6003.932,E2 -6003.932} C_VEL
LIN {X 0,Y 495.759,Z 196.044,A -85,B 0,C 180,E1 -6007.139,E2 -6007.139} C_VEL
LIN {X 0,Y 495.77,Z 196.032,A -85,B 0,C 180,E1 -6010.11,E2 -6010.11} C_VEL
LIN {X 0,Y 495.764,Z 196.039,A -85,B 0,C 180,E1 -6012.681,E2 -6012.681} C_VEL
LIN {X 0,Y 495.789,Z 196.032,A -85,B 0,C 180,E1 -6015.217,E2 -6015.217} C_VEL
LIN {X 0,Y 495.851,Z 196.033,A -85,B 0,C 180,E1 -6018.555,E2 -6018.555} C_VEL
LIN {X 0,Y 495.873,Z 196.028,A -85,B 0,C 180,E1 -6021.852,E2 -6021.852} C_VEL
LIN {X 0,Y 495.838,Z 196.036,A -85,B 0,C 180,E1 -6025.121,E2 -6025.121} C_VEL
LIN {X 0,Y 495.907,Z 196.095,A -85,B 0,C 180,E1 -6026.928,E2 -6026.928} C_VEL
LIN {X 0,Y 499.316,Z 207.99,A -85,B 0,C 180,E1 -6028.535,E2 -6028.535} C_VEL
LIN {X 0,Y 504.228,Z 219.043,A -85,B 0,C 180,E1 -6029.001,E2 -6029.001} C_VEL
LIN {X 0,Y 505.487,Z 225.651,A -85,B 0,C 180,E1 -6029.178,E2 -6029.178} C_VEL
LIN {X 0,Y 503.301,Z 414.203,A -85,B 0,C 180,E1 -6032.025,E2 -6032.025} C_VEL
LIN {X 0,Y 502.887,Z 431.069,A -85,B 0,C 180,E1 -6032.453,E2 -6032.453} C_VEL
LIN {X 0,Y 502.253,Z 446.812,A -85,B 0,C 180,E1 -6033.008,E2 -6033.008} C_VEL
LIN {X 0,Y 501.563,Z 462.264,A -85,B 0,C 180,E1 -6033.715,E2 -6033.715} C_VEL
LIN {X 0,Y 500.829,Z 476.455,A -85,B 0,C 180,E1 -6034.516,E2 -6034.516} C_VEL
LIN {X 0,Y 499.962,Z 491.351,A -85,B 0,C 180,E1 -6035.546,E2 -6035.546} C_VEL
LIN {X 0,Y 499.144,Z 504.911,A -85,B 0,C 180,E1 -6036.67,E2 -6036.67} C_VEL
LIN {X 0,Y 498.302,Z 517.566,A -85,B 0,C 180,E1 -6037.904,E2 -6037.904} C_VEL
LIN {X 0,Y 497.579,Z 528.519,A -85,B 0,C 180,E1 -6039.143,E2 -6039.143} C_VEL
LIN {X 0,Y 496.896,Z 539.441,A -85,B 0,C 180,E1 -6040.595,E2 -6040.595} C_VEL
LIN {X 0,Y 496.341,Z 549.329,A -85,B 0,C 180,E1 -6042.137,E2 -6042.137} C_VEL
LIN {X 0,Y 495.857,Z 558.046,A -85,B 0,C 180,E1 -6043.733,E2 -6043.733} C_VEL
LIN {X 0,Y 495.522,Z 565.346,A -85,B 0,C 180,E1 -6045.325,E2 -6045.325} C_VEL
LIN {X 0,Y 495.292,Z 571.387,A -85,B 0,C 180,E1 -6046.911,E2 -6046.911} C_VEL
LIN {X 0,Y 495.146,Z 576.742,A -85,B 0,C 180,E1 -6048.624,E2 -6048.624} C_VEL
LIN {X 0,Y 495.015,Z 581.071,A -85,B 0,C 180,E1 -6050.441,E2 -6050.441} C_VEL
LIN {X 0,Y 494.91,Z 583.312,A -85,B 0,C 180,E1 -6051.667,E2 -6051.667} C_VEL
LIN {X 0,Y 494.835,Z 585.491,A -85,B 0,C 180,E1 -6053.432,E2 -6053.432} C_VEL
LIN {X 0,Y 494.849,Z 586.599,A -85,B 0,C 180,E1 -6055.218,E2 -6055.218} C_VEL
LIN {X 0,Y 494.879,Z 586.572,A -85,B 0,C 180,E1 -6057.029,E2 -6057.029} C_VEL
LIN {X 0,Y 494.903,Z 585.295,A -85,B 0,C 180,E1 -6058.869,E2 -6058.869} C_VEL
LIN {X 0,Y 494.959,Z 582.776,A -85,B 0,C 180,E1 -6060.741,E2 -6060.741} C_VEL
LIN {X 0,Y 495.063,Z 578.882,A -85,B 0,C 180,E1 -6062.646,E2 -6062.646} C_VEL
LIN {X 0,Y 495.264,Z 573.455,A -85,B 0,C 180,E1 -6064.583,E2 -6064.583} C_VEL
LIN {X 0,Y 495.421,Z 567.398,A -85,B 0,C 180,E1 -6066.269,E2 -6066.269} C_VEL
LIN {X 0,Y 495.795,Z 559.502,A -85,B 0,C 180,E1 -6068.069,E2 -6068.069} C_VEL
LIN {X 0,Y 496.201,Z 551.52,A -85,B 0,C 180,E1 -6069.594,E2 -6069.594} C_VEL
LIN {X 0,Y 496.829,Z 540.994,A -85,B 0,C 180,E1 -6071.286,E2 -6071.286} C_VEL
LIN {X 0,Y 497.47,Z 530.374,A -85,B 0,C 180,E1 -6072.724,E2 -6072.724} C_VEL
LIN {X 0,Y 498.272,Z 518.437,A -85,B 0,C 180,E1 -6074.104,E2 -6074.104} C_VEL
LIN {X 0,Y 499.119,Z 505.599,A -85,B 0,C 180,E1 -6075.369,E2 -6075.369} C_VEL
LIN {X 0,Y 499.913,Z 492.617,A -85,B 0,C 180,E1 -6076.46,E2 -6076.46} C_VEL
LIN {X 0,Y 500.716,Z 478.791,A -85,B 0,C 180,E1 -6077.429,E2 -6077.429} C_VEL
LIN {X 0,Y 501.475,Z 464.442,A -85,B 0,C 180,E1 -6078.268,E2 -6078.268} C_VEL
LIN {X 0,Y 502.227,Z 448.5,A -85,B 0,C 180,E1 -6079.019,E2 -6079.019} C_VEL
LIN {X 0,Y 502.807,Z 433.172,A -85,B 0,C 180,E1 -6079.581,E2 -6079.581} C_VEL
LIN {X 0,Y 503.29,Z 416.301,A -85,B 0,C 180,E1 -6080.02,E2 -6080.02} C_VEL
LIN {X 0,Y 503.628,Z 389.658,A -85,B 0,C 180,E1 -6080.455,E2 -6080.455} C_VEL
LIN {X 0,Y 505.454,Z 224.857,A -85,B 0,C 180,E1 -6082.939,E2 -6082.939} C_VEL
LIN {X 0,Y 504.005,Z 218.596,A -85,B 0,C 180,E1 -6083.124,E2 -6083.124} C_VEL
LIN {X 0,Y 499.284,Z 208.157,A -85,B 0,C 180,E1 -6083.591,E2 -6083.591} C_VEL
LIN {X 0,Y 495.757,Z 196.047,A -85,B 0,C 180,E1 -6085.275,E2 -6085.275} C_VEL
LIN {X 0,Y 495.746,Z 196.047,A -85,B 0,C 180,E1 -6088.363,E2 -6088.363} C_VEL
LIN {X 0,Y 495.747,Z 196.047,A -85,B 0,C 180,E1 -6091.514,E2 -6091.514} C_VEL
LIN {X 0,Y 495.71,Z 196.048,A -85,B 0,C 180,E1 -6093.928,E2 -6093.928} C_VEL
LIN {X 0,Y 495.75,Z 196.044,A -85,B 0,C 180,E1 -6097.14,E2 -6097.14} C_VEL
LIN {X 0,Y 495.762,Z 196.042,A -85,B 0,C 180,E1 -6100.109,E2 -6100.109} C_VEL
LIN {X 0,Y 495.756,Z 196.048,A -85,B 0,C 180,E1 -6102.68,E2 -6102.68} C_VEL
LIN {X 0,Y 495.782,Z 196.04,A -85,B 0,C 180,E1 -6105.217,E2 -6105.217} C_VEL
LIN {X 0,Y 495.844,Z 196.029,A -85,B 0,C 180,E1 -6108.555,E2 -6108.555} C_VEL
LIN {X 0,Y 495.829,Z 196.032,A -85,B 0,C 180,E1 -6111.851,E2 -6111.851} C_VEL
LIN {X 0,Y 495.88,Z 196.03,A -85,B 0,C 180,E1 -6114.306,E2 -6114.306} C_VEL
LIN {X 0,Y 495.984,Z 196.012,A -85,B 0,C 180,E1 -6117.564,E2 -6117.564} C_VEL
LIN {X 0,Y 495.99,Z 196.016,A -85,B 0,C 180,E1 -6120,E2 -6120} C_VEL
LIN {X 0,Y 495.986,Z 196.015,A -85,B 0,C 180,E1 -6122.436,E2 -6122.436} C_VEL
LIN {X 0,Y 495.888,Z 196.026,A -85,B 0,C 180,E1 -6125.694,E2 -6125.694} C_VEL
LIN {X 0,Y 495.866,Z 196.031,A -85,B 0,C 180,E1 -6128.148,E2 -6128.148} C_VEL
LIN {X 0,Y 495.845,Z 196.029,A -85,B 0,C 180,E1 -6131.445,E2 -6131.445} C_VEL
LIN {X 0,Y 495.783,Z 196.037,A -85,B 0,C 180,E1 -6134.783,E2 -6134.783} C_VEL
LIN {X 0,Y 495.781,Z 196.038,A -85,B 0,C 180,E1 -6137.319,E2 -6137.319} C_VEL
LIN {X 0,Y 495.766,Z 196.046,A -85,B 0,C 180,E1 -6139.89,E2 -6139.89} C_VEL
LIN {X 0,Y 495.759,Z 196.04,A -85,B 0,C 180,E1 -6142.863,E2 -6142.863} C_VEL
LIN {X 0,Y 495.793,Z 196.037,A -85,B 0,C 180,E1 -6146.068,E2 -6146.068} C_VEL
LIN {X 0,Y 495.766,Z 196.04,A -85,B 0,C 180,E1 -6148.815,E2 -6148.815} C_VEL
LIN {X 0,Y 495.753,Z 196.047,A -85,B 0,C 180,E1 -6151.726,E2 -6151.726} C_VEL
LIN {X 0,Y 495.766,Z 196.042,A -85,B 0,C 180,E1 -6154.695,E2 -6154.695} C_VEL
LIN {X 0,Y 495.723,Z 196.051,A -85,B 0,C 180,E1 -6157.562,E2 -6157.562} C_VEL
LIN {X 0,Y 495.761,Z 196.044,A -85,B 0,C 180,E1 -6160.7,E2 -6160.7} C_VEL
LIN {X 0,Y 495.729,Z 196.047,A -85,B 0,C 180,E1 -6164.001,E2 -6164.001} C_VEL
LIN {X 0,Y 495.72,Z 196.053,A -85,B 0,C 180,E1 -6167.117,E2 -6167.117} C_VEL
LIN {X 0,Y 495.754,Z 196.043,A -85,B 0,C 180,E1 -6169.953,E2 -6169.953} C_VEL
LIN {X 0,Y 495.723,Z 196.049,A -85,B 0,C 180,E1 -6172.554,E2 -6172.554} C_VEL
LIN {X 0,Y 495.773,Z 196.04,A -85,B 0,C 180,E1 -6175.457,E2 -6175.457} C_VEL
LIN {X 0,Y 495.764,Z 196.072,A -85,B 0,C 180,E1 -6178.389,E2 -6178.389} C_VEL
LIN {X 0,Y 501.744,Z 215.91,A -85,B 0,C 180,E1 -6180.874,E2 -6180.874} C_VEL
LIN {X 0,Y 502.375,Z 218.141,A -85,B 0,C 180,E1 -6181.143,E2 -6181.143} C_VEL
LIN {X 0,Y 501.67,Z 232.882,A -85,B 0,C 180,E1 -6182.605,E2 -6182.605} C_VEL
LIN {X 0,Y 505.337,Z 253.421,A -85,B 0,C 180,E1 -6183.146,E2 -6183.146} C_VEL
LIN {X 0,Y 503.198,Z 438.968,A -85,B 0,C 180,E1 -6185.943,E2 -6185.943} C_VEL
LIN {X 0,Y 502.703,Z 455.278,A -85,B 0,C 180,E1 -6186.329,E2 -6186.329} C_VEL
LIN {X 0,Y 502.123,Z 471.471,A -85,B 0,C 180,E1 -6186.873,E2 -6186.873} C_VEL
LIN {X 0,Y 501.39,Z 486.884,A -85,B 0,C 180,E1 -6187.546,E2 -6187.546} C_VEL
LIN {X 0,Y 500.596,Z 502.41,A -85,B 0,C 180,E1 -6188.403,E2 -6188.403} C_VEL
LIN {X 0,Y 499.686,Z 517.369,A -85,B 0,C 180,E1 -6189.414,E2 -6189.414} C_VEL
LIN {X 0,Y 498.84,Z 531.189,A -85,B 0,C 180,E1 -6190.533,E2 -6190.533} C_VEL
LIN {X 0,Y 498.067,Z 543.53,A -85,B 0,C 180,E1 -6191.702,E2 -6191.702} C_VEL
LIN {X 0,Y 497.366,Z 554.822,A -85,B 0,C 180,E1 -6192.95,E2 -6192.95} C_VEL
LIN {X 0,Y 496.707,Z 566.097,A -85,B 0,C 180,E1 -6194.406,E2 -6194.406} C_VEL
LIN {X 0,Y 496.175,Z 575.773,A -85,B 0,C 180,E1 -6195.858,E2 -6195.858} C_VEL
LIN {X 0,Y 495.798,Z 585.179,A -85,B 0,C 180,E1 -6197.516,E2 -6197.516} C_VEL
LIN {X 0,Y 495.44,Z 593.886,A -85,B 0,C 180,E1 -6199.374,E2 -6199.374} C_VEL
LIN {X 0,Y 495.164,Z 601.599,A -85,B 0,C 180,E1 -6201.43,E2 -6201.43} C_VEL
LIN {X 0,Y 495.11,Z 606.387,A -85,B 0,C 180,E1 -6203.07,E2 -6203.07} C_VEL
LIN {X 0,Y 495.034,Z 609.302,A -85,B 0,C 180,E1 -6204.297,E2 -6204.297} C_VEL
LIN {X 0,Y 494.973,Z 612.261,A -85,B 0,C 180,E1 -6205.929,E2 -6205.929} C_VEL
LIN {X 0,Y 494.991,Z 614.21,A -85,B 0,C 180,E1 -6207.559,E2 -6207.559} C_VEL
LIN {X 0,Y 494.907,Z 615.176,A -85,B 0,C 180,E1 -6209.187,E2 -6209.187} C_VEL
LIN {X 0,Y 494.907,Z 615.179,A -85,B 0,C 180,E1 -6210.814,E2 -6210.814} C_VEL
LIN {X 0,Y 494.991,Z 614.218,A -85,B 0,C 180,E1 -6212.441,E2 -6212.441} C_VEL
LIN {X 0,Y 494.973,Z 612.276,A -85,B 0,C 180,E1 -6214.071,E2 -6214.071} C_VEL
LIN {X 0,Y 495.034,Z 609.326,A -85,B 0,C 180,E1 -6215.704,E2 -6215.704} C_VEL
LIN {X 0,Y 495.139,Z 605.343,A -85,B 0,C 180,E1 -6217.339,E2 -6217.339} C_VEL
LIN {X 0,Y 495.205,Z 600.205,A -85,B 0,C 180,E1 -6218.981,E2 -6218.981} C_VEL
LIN {X 0,Y 495.446,Z 593.937,A -85,B 0,C 180,E1 -6220.627,E2 -6220.627} C_VEL
LIN {X 0,Y 495.818,Z 585.246,A -85,B 0,C 180,E1 -6222.484,E2 -6222.484} C_VEL
LIN {X 0,Y 496.179,Z 575.858,A -85,B 0,C 180,E1 -6224.142,E2 -6224.142} C_VEL
LIN {X 0,Y 496.717,Z 566.199,A -85,B 0,C 180,E1 -6225.595,E2 -6225.595} C_VEL
LIN {X 0,Y 497.388,Z 554.942,A -85,B 0,C 180,E1 -6227.049,E2 -6227.049} C_VEL
LIN {X 0,Y 498.14,Z 542.685,A -85,B 0,C 180,E1 -6228.402,E2 -6228.402} C_VEL
LIN {X 0,Y 499.051,Z 528.099,A -85,B 0,C 180,E1 -6229.754,E2 -6229.754} C_VEL
LIN {X 0,Y 499.953,Z 513.251,A -85,B 0,C 180,E1 -6230.898,E2 -6230.898} C_VEL
LIN {X 0,Y 500.761,Z 499.465,A -85,B 0,C 180,E1 -6231.782,E2 -6231.782} C_VEL
LIN {X 0,Y 501.613,Z 483.587,A -85,B 0,C 180,E1 -6232.619,E2 -6232.619} C_VEL
LIN {X 0,Y 502.264,Z 469.127,A -85,B 0,C 180,E1 -6233.23,E2 -6233.23} C_VEL
LIN {X 0,Y 502.79,Z 452.822,A -85,B 0,C 180,E1 -6233.75,E2 -6233.75} C_VEL
LIN {X 0,Y 503.276,Z 436.298,A -85,B 0,C 180,E1 -6234.108,E2 -6234.108} C_VEL
LIN {X 0,Y 505.326,Z 253.759,A -85,B 0,C 180,E1 -6236.85,E2 -6236.85} C_VEL
LIN {X 0,Y 501.71,Z 233.073,A -85,B 0,C 180,E1 -6237.395,E2 -6237.395} C_VEL
LIN {X 0,Y 502.434,Z 218.395,A -85,B 0,C 180,E1 -6238.854,E2 -6238.854} C_VEL
LIN {X 0,Y 496.865,Z 199.786,A -85,B 0,C 180,E1 -6241.152,E2 -6241.152} C_VEL
LIN {X 0,Y 495.752,Z 196.042,A -85,B 0,C 180,E1 -6241.636,E2 -6241.636} C_VEL
LIN {X 0,Y 495.774,Z 196.042,A -85,B 0,C 180,E1 -6244.543,E2 -6244.543} C_VEL
LIN {X 0,Y 495.719,Z 196.048,A -85,B 0,C 180,E1 -6247.562,E2 -6247.562} C_VEL
LIN {X 0,Y 495.754,Z 196.038,A -85,B 0,C 180,E1 -6250.047,E2 -6250.047} C_VEL
LIN {X 0,Y 495.714,Z 196.048,A -85,B 0,C 180,E1 -6252.884,E2 -6252.884} C_VEL
LIN {X 0,Y 495.72,Z 196.041,A -85,B 0,C 180,E1 -6255.998,E2 -6255.998} C_VEL
LIN {X 0,Y 495.737,Z 196.047,A -85,B 0,C 180,E1 -6258.709,E2 -6258.709} C_VEL
LIN {X 0,Y 495.744,Z 196.045,A -85,B 0,C 180,E1 -6261.408,E2 -6261.408} C_VEL
LIN {X 0,Y 495.743,Z 196.039,A -85,B 0,C 180,E1 -6264.462,E2 -6264.462} C_VEL
LIN {X 0,Y 495.763,Z 196.036,A -85,B 0,C 180,E1 -6267.405,E2 -6267.405} C_VEL
LIN {X 0,Y 495.762,Z 196.04,A -85,B 0,C 180,E1 -6270.254,E2 -6270.254} C_VEL
LIN {X 0,Y 495.82,Z 196.026,A -85,B 0,C 180,E1 -6273.251,E2 -6273.251} C_VEL
LIN {X 0,Y 495.739,Z 196.048,A -85,B 0,C 180,E1 -6276.612,E2 -6276.612} C_VEL
LIN {X 0,Y 495.775,Z 196.033,A -85,B 0,C 180,E1 -6279.324,E2 -6279.324} C_VEL
LIN {X 0,Y 495.775,Z 196.03,A -85,B 0,C 180,E1 -6281.828,E2 -6281.828} C_VEL
LIN {X 0,Y 495.82,Z 196.039,A -85,B 0,C 180,E1 -6284.548,E2 -6284.548} C_VEL
LIN {X 0,Y 495.825,Z 196.023,A -85,B 0,C 180,E1 -6287.965,E2 -6287.965} C_VEL
LIN {X 0,Y 495.833,Z 196.031,A -85,B 0,C 180,E1 -6291.03,E2 -6291.03} C_VEL
LIN {X 0,Y 495.856,Z 196.027,A -85,B 0,C 180,E1 -6293.489,E2 -6293.489} C_VEL
LIN {X 0,Y 495.837,Z 196.015,A -85,B 0,C 180,E1 -6296.75,E2 -6296.75} C_VEL
LIN {X 0,Y 495.868,Z 196.02,A -85,B 0,C 180,E1 -6298.376,E2 -6298.376} C_VEL
LIN {X 0,Y 496.001,Z 196.011,A -85,B 0,C 180,E1 -6300.812,E2 -6300.812} C_VEL
LIN {X 0,Y 495.837,Z 196.028,A -85,B 0,C 180,E1 -6303.25,E2 -6303.25} C_VEL
LIN {X 0,Y 495.875,Z 196.027,A -85,B 0,C 180,E1 -6306.51,E2 -6306.51} C_VEL
LIN {X 0,Y 495.835,Z 196.029,A -85,B 0,C 180,E1 -6308.97,E2 -6308.97} C_VEL
LIN {X 0,Y 495.825,Z 196.029,A -85,B 0,C 180,E1 -6312.035,E2 -6312.035} C_VEL
LIN {X 0,Y 495.821,Z 196.033,A -85,B 0,C 180,E1 -6315.452,E2 -6315.452} C_VEL
LIN {X 0,Y 495.804,Z 196.029,A -85,B 0,C 180,E1 -6318.247,E2 -6318.247} C_VEL
LIN {X 0,Y 495.771,Z 196.036,A -85,B 0,C 180,E1 -6320.756,E2 -6320.756} C_VEL
LIN {X 0,Y 495.749,Z 196.042,A -85,B 0,C 180,E1 -6323.387,E2 -6323.387} C_VEL
LIN {X 0,Y 495.788,Z 196.036,A -85,B 0,C 180,E1 -6326.068,E2 -6326.068} C_VEL
LIN {X 0,Y 495.776,Z 196.037,A -85,B 0,C 180,E1 -6328.814,E2 -6328.814} C_VEL
LIN {X 0,Y 495.754,Z 196.039,A -85,B 0,C 180,E1 -6331.726,E2 -6331.726} C_VEL
LIN {X 0,Y 495.774,Z 196.037,A -85,B 0,C 180,E1 -6334.695,E2 -6334.695} C_VEL
LIN {X 0,Y 495.729,Z 196.044,A -85,B 0,C 180,E1 -6337.562,E2 -6337.562} C_VEL
LIN {X 0,Y 495.764,Z 196.039,A -85,B 0,C 180,E1 -6340.7,E2 -6340.7} C_VEL
LIN {X 0,Y 495.725,Z 196.042,A -85,B 0,C 180,E1 -6344.002,E2 -6344.002} C_VEL
LIN {X 0,Y 495.723,Z 196.048,A -85,B 0,C 180,E1 -6347.117,E2 -6347.117} C_VEL
LIN {X 0,Y 495.756,Z 196.041,A -85,B 0,C 180,E1 -6349.953,E2 -6349.953} C_VEL
LIN {X 0,Y 495.726,Z 196.043,A -85,B 0,C 180,E1 -6352.553,E2 -6352.553} C_VEL
LIN {X 0,Y 495.779,Z 196.044,A -85,B 0,C 180,E1 -6355.457,E2 -6355.457} C_VEL
LIN {X 0,Y 495.755,Z 196.036,A -85,B 0,C 180,E1 -6358.364,E2 -6358.364} C_VEL
LIN {X 0,Y 495.752,Z 196.043,A -85,B 0,C 180,E1 -6360.761,E2 -6360.761} C_VEL
LIN {X 0,Y 495.096,Z 196.13,A -85,B 0,C 180,E1 -6361.44,E2 -6361.44} C_VEL
LIN {X 0,Y 492.239,Z 196.483,A -85,B 0,C 180,E1 -6362.543,E2 -6362.543} C_VEL
LIN {X 0,Y 489.83,Z 196.783,A -85,B 0,C 180,E1 -6363.432,E2 -6363.432} C_VEL
LIN {X 0,Y 488.814,Z 196.906,A -85,B 0,C 180,E1 -6364.118,E2 -6364.118} C_VEL
LIN {X 0,Y 488.742,Z 196.914,A -85,B 0,C 180,E1 -6364.35,E2 -6364.35} C_VEL
LIN {X 0,Y 488.722,Z 196.92,A -85,B 0,C 180,E1 -6367.153,E2 -6367.153} C_VEL
LIN {X 0,Y 488.724,Z 196.91,A -85,B 0,C 180,E1 -6369.81,E2 -6369.81} C_VEL
LIN {X 0,Y 488.714,Z 196.915,A -85,B 0,C 180,E1 -6372.423,E2 -6372.423} C_VEL
LIN {X 0,Y 488.761,Z 196.911,A -85,B 0,C 180,E1 -6375,E2 -6375} C_VEL
LIN {X 0,Y 488.805,Z 196.909,A -85,B 0,C 180,E1 -6378.387,E2 -6378.387} C_VEL
LIN {X 0,Y 488.817,Z 196.908,A -85,B 0,C 180,E1 -6381.733,E2 -6381.733} C_VEL
LIN {X 0,Y 488.808,Z 196.912,A -85,B 0,C 180,E1 -6385.051,E2 -6385.051} C_VEL
LIN {X 0,Y 488.78,Z 196.965,A -85,B 0,C 180,E1 -6386.548,E2 -6386.548} C_VEL
LIN {X 0,Y 492.118,Z 208.321,A -85,B 0,C 180,E1 -6388.103,E2 -6388.103} C_VEL
LIN {X 0,Y 498.192,Z 221.773,A -85,B 0,C 180,E1 -6388.69,E2 -6388.69} C_VEL
LIN {X 0,Y 499.155,Z 226.595,A -85,B 0,C 180,E1 -6388.825,E2 -6388.825} C_VEL
LIN {X 0,Y 496.824,Z 414.411,A -85,B 0,C 180,E1 -6391.697,E2 -6391.697} C_VEL
LIN {X 0,Y 496.38,Z 431.29,A -85,B 0,C 180,E1 -6392.13,E2 -6392.13} C_VEL
LIN {X 0,Y 495.718,Z 447.027,A -85,B 0,C 180,E1 -6392.691,E2 -6392.691} C_VEL
LIN {X 0,Y 494.928,Z 463.455,A -85,B 0,C 180,E1 -6393.46,E2 -6393.46} C_VEL
LIN {X 0,Y 494.077,Z 478.808,A -85,B 0,C 180,E1 -6394.361,E2 -6394.361} C_VEL
LIN {X 0,Y 493.235,Z 492.279,A -85,B 0,C 180,E1 -6395.314,E2 -6395.314} C_VEL
LIN {X 0,Y 492.254,Z 506.894,A -85,B 0,C 180,E1 -6396.558,E2 -6396.558} C_VEL
LIN {X 0,Y 491.387,Z 519.252,A -85,B 0,C 180,E1 -6397.809,E2 -6397.809} C_VEL
LIN {X 0,Y 490.52,Z 531.603,A -85,B 0,C 180,E1 -6399.275,E2 -6399.275} C_VEL
LIN {X 0,Y 489.808,Z 542.182,A -85,B 0,C 180,E1 -6400.75,E2 -6400.75} C_VEL
LIN {X 0,Y 489.223,Z 552.449,A -85,B 0,C 180,E1 -6402.444,E2 -6402.444} C_VEL
LIN {X 0,Y 488.729,Z 561.075,A -85,B 0,C 180,E1 -6404.15,E2 -6404.15} C_VEL
LIN {X 0,Y 488.342,Z 568.295,A -85,B 0,C 180,E1 -6405.869,E2 -6405.869} C_VEL
LIN {X 0,Y 488.169,Z 574.258,A -85,B 0,C 180,E1 -6407.597,E2 -6407.597} C_VEL
LIN {X 0,Y 488.027,Z 579.038,A -85,B 0,C 180,E1 -6409.342,E2 -6409.342} C_VEL
LIN {X 0,Y 487.854,Z 582.659,A -85,B 0,C 180,E1 -6411.109,E2 -6411.109} C_VEL
LIN {X 0,Y 487.77,Z 585.211,A -85,B 0,C 180,E1 -6412.893,E2 -6412.893} C_VEL
LIN {X 0,Y 487.756,Z 586.673,A -85,B 0,C 180,E1 -6414.803,E2 -6414.803} C_VEL
LIN {X 0,Y 487.78,Z 586.84,A -85,B 0,C 180,E1 -6416.709,E2 -6416.709} C_VEL
LIN {X 0,Y 487.817,Z 585.892,A -85,B 0,C 180,E1 -6418.499,E2 -6418.499} C_VEL
LIN {X 0,Y 487.862,Z 583.839,A -85,B 0,C 180,E1 -6420.278,E2 -6420.278} C_VEL
LIN {X 0,Y 488.011,Z 580.305,A -85,B 0,C 180,E1 -6422.197,E2 -6422.197} C_VEL
LIN {X 0,Y 488.153,Z 575.29,A -85,B 0,C 180,E1 -6424.158,E2 -6424.158} C_VEL
LIN {X 0,Y 488.303,Z 570.474,A -85,B 0,C 180,E1 -6425.654,E2 -6425.654} C_VEL
LIN {X 0,Y 488.605,Z 563.359,A -85,B 0,C 180,E1 -6427.445,E2 -6427.445} C_VEL
LIN {X 0,Y 489.037,Z 554.791,A -85,B 0,C 180,E1 -6429.221,E2 -6429.221} C_VEL
LIN {X 0,Y 489.635,Z 545.519,A -85,B 0,C 180,E1 -6430.832,E2 -6430.832} C_VEL
LIN {X 0,Y 490.283,Z 535.249,A -85,B 0,C 180,E1 -6432.354,E2 -6432.354} C_VEL
LIN {X 0,Y 491.138,Z 523.624,A -85,B 0,C 180,E1 -6433.806,E2 -6433.806} C_VEL
LIN {X 0,Y 491.953,Z 511.031,A -85,B 0,C 180,E1 -6435.148,E2 -6435.148} C_VEL
LIN {X 0,Y 492.867,Z 497.972,A -85,B 0,C 180,E1 -6436.327,E2 -6436.327} C_VEL
LIN {X 0,Y 493.75,Z 484.693,A -85,B 0,C 180,E1 -6437.348,E2 -6437.348} C_VEL
LIN {X 0,Y 494.624,Z 470.024,A -85,B 0,C 180,E1 -6438.28,E2 -6438.28} C_VEL
LIN {X 0,Y 495.405,Z 454.668,A -85,B 0,C 180,E1 -6439.075,E2 -6439.075} C_VEL
LIN {X 0,Y 496.094,Z 438.327,A -85,B 0,C 180,E1 -6439.737,E2 -6439.737} C_VEL
LIN {X 0,Y 496.681,Z 422.225,A -85,B 0,C 180,E1 -6440.218,E2 -6440.218} C_VEL
LIN {X 0,Y 497.021,Z 405.778,A -85,B 0,C 180,E1 -6440.549,E2 -6440.549} C_VEL
LIN {X 0,Y 499.16,Z 226.268,A -85,B 0,C 180,E1 -6443.29,E2 -6443.29} C_VEL
LIN {X 0,Y 498.034,Z 221.357,A -85,B 0,C 180,E1 -6443.437,E2 -6443.437} C_VEL
LIN {X 0,Y 492.101,Z 208.42,A -85,B 0,C 180,E1 -6444.032,E2 -6444.032} C_VEL
LIN {X 0,Y 488.714,Z 196.922,A -85,B 0,C 180,E1 -6445.668,E2 -6445.668} C_VEL
LIN {X 0,Y 488.683,Z 196.928,A -85,B 0,C 180,E1 -6448.82,E2 -6448.82} C_VEL
LIN {X 0,Y 488.703,Z 196.923,A -85,B 0,C 180,E1 -6451.669,E2 -6451.669} C_VEL
LIN {X 0,Y 488.691,Z 196.924,A -85,B 0,C 180,E1 -6454.959,E2 -6454.959} C_VEL
LIN {X 0,Y 488.689,Z 196.918,A -85,B 0,C 180,E1 -6458.043,E2 -6458.043} C_VEL
LIN {X 0,Y 488.734,Z 196.918,A -85,B 0,C 180,E1 -6460.686,E2 -6460.686} C_VEL
LIN {X 0,Y 488.754,Z 196.913,A -85,B 0,C 180,E1 -6464.145,E2 -6464.145} C_VEL
LIN {X 0,Y 488.723,Z 196.921,A -85,B 0,C 180,E1 -6466.698,E2 -6466.698} C_VEL
LIN {X 0,Y 488.731,Z 196.917,A -85,B 0,C 180,E1 -6469.226,E2 -6469.226} C_VEL
LIN {X 0,Y 488.778,Z 196.91,A -85,B 0,C 180,E1 -6471.733,E2 -6471.733} C_VEL
LIN {X 0,Y 488.839,Z 196.906,A -85,B 0,C 180,E1 -6474.224,E2 -6474.224} C_VEL
LIN {X 0,Y 488.952,Z 196.888,A -85,B 0,C 180,E1 -6477.529,E2 -6477.529} C_VEL
LIN {X 0,Y 488.948,Z 196.89,A -85,B 0,C 180,E1 -6480.824,E2 -6480.824} C_VEL
LIN {X 0,Y 488.953,Z 196.891,A -85,B 0,C 180,E1 -6482.471,E2 -6482.471} C_VEL
LIN {X 0,Y 488.847,Z 196.904,A -85,B 0,C 180,E1 -6485.776,E2 -6485.776} C_VEL
LIN {X 0,Y 488.811,Z 196.91,A -85,B 0,C 180,E1 -6488.266,E2 -6488.266} C_VEL
LIN {X 0,Y 488.799,Z 196.908,A -85,B 0,C 180,E1 -6491.613,E2 -6491.613} C_VEL
LIN {X 0,Y 488.755,Z 196.913,A -85,B 0,C 180,E1 -6495.001,E2 -6495.001} C_VEL
LIN {X 0,Y 488.748,Z 196.913,A -85,B 0,C 180,E1 -6498.442,E2 -6498.442} C_VEL
LIN {X 0,Y 488.7,Z 196.92,A -85,B 0,C 180,E1 -6501.071,E2 -6501.071} C_VEL
LIN {X 0,Y 488.688,Z 196.926,A -85,B 0,C 180,E1 -6503.746,E2 -6503.746} C_VEL
LIN {X 0,Y 488.793,Z 196.907,A -85,B 0,C 180,E1 -6506.946,E2 -6506.946} C_VEL
LIN {X 0,Y 488.704,Z 196.92,A -85,B 0,C 180,E1 -6510.363,E2 -6510.363} C_VEL
LIN {X 0,Y 488.73,Z 196.922,A -85,B 0,C 180,E1 -6513.485,E2 -6513.485} C_VEL
LIN {X 0,Y 488.677,Z 196.925,A -85,B 0,C 180,E1 -6516.355,E2 -6516.355} C_VEL
LIN {X 0,Y 488.696,Z 196.93,A -85,B 0,C 180,E1 -6519.255,E2 -6519.255} C_VEL
LIN {X 0,Y 488.702,Z 196.925,A -85,B 0,C 180,E1 -6521.6,E2 -6521.6} C_VEL
LIN {X 0,Y 488.707,Z 196.926,A -85,B 0,C 180,E1 -6524.802,E2 -6524.802} C_VEL
LIN {X 0,Y 488.686,Z 196.928,A -85,B 0,C 180,E1 -6527.475,E2 -6527.475} C_VEL
LIN {X 0,Y 488.728,Z 196.919,A -85,B 0,C 180,E1 -6529.677,E2 -6529.677} C_VEL
LIN {X 0,Y 488.675,Z 196.929,A -85,B 0,C 180,E1 -6532.842,E2 -6532.842} C_VEL
LIN {X 0,Y 488.726,Z 196.916,A -85,B 0,C 180,E1 -6535.888,E2 -6535.888} C_VEL
LIN {X 0,Y 488.704,Z 196.923,A -85,B 0,C 180,E1 -6537.987,E2 -6537.987} C_VEL
LIN {X 0,Y 494.679,Z 216.647,A -85,B 0,C 180,E1 -6540.514,E2 -6540.514} C_VEL
LIN {X 0,Y 495.766,Z 220.528,A -85,B 0,C 180,E1 -6540.989,E2 -6540.989} C_VEL
LIN {X 0,Y 495.101,Z 232.423,A -85,B 0,C 180,E1 -6542.19,E2 -6542.19} C_VEL
LIN {X 0,Y 498.987,Z 255.022,A -85,B 0,C 180,E1 -6542.802,E2 -6542.802} C_VEL
LIN {X 0,Y 496.722,Z 438.885,A -85,B 0,C 180,E1 -6545.614,E2 -6545.614} C_VEL
LIN {X 0,Y 496.199,Z 454.986,A -85,B 0,C 180,E1 -6545.999,E2 -6545.999} C_VEL
LIN {X 0,Y 495.568,Z 471.189,A -85,B 0,C 180,E1 -6546.549,E2 -6546.549} C_VEL
LIN {X 0,Y 494.805,Z 486.602,A -85,B 0,C 180,E1 -6547.23,E2 -6547.23} C_VEL
LIN {X 0,Y 493.932,Z 502.382,A -85,B 0,C 180,E1 -6548.112,E2 -6548.112} C_VEL
LIN {X 0,Y 493.061,Z 515.667,A -85,B 0,C 180,E1 -6549.015,E2 -6549.015} C_VEL
LIN {X 0,Y 492.11,Z 530.095,A -85,B 0,C 180,E1 -6550.179,E2 -6550.179} C_VEL
LIN {X 0,Y 491.203,Z 543.279,A -85,B 0,C 180,E1 -6551.438,E2 -6551.438} C_VEL
LIN {X 0,Y 490.446,Z 554.574,A -85,B 0,C 180,E1 -6552.702,E2 -6552.702} C_VEL
LIN {X 0,Y 489.731,Z 565.856,A -85,B 0,C 180,E1 -6554.178,E2 -6554.178} C_VEL
LIN {X 0,Y 489.169,Z 575.538,A -85,B 0,C 180,E1 -6555.651,E2 -6555.651} C_VEL
LIN {X 0,Y 488.771,Z 584.95,A -85,B 0,C 180,E1 -6557.334,E2 -6557.334} C_VEL
LIN {X 0,Y 488.374,Z 593.661,A -85,B 0,C 180,E1 -6559.218,E2 -6559.218} C_VEL
LIN {X 0,Y 488.089,Z 601.381,A -85,B 0,C 180,E1 -6561.304,E2 -6561.304} C_VEL
LIN {X 0,Y 487.994,Z 607.254,A -85,B 0,C 180,E1 -6563.384,E2 -6563.384} C_VEL
LIN {X 0,Y 487.907,Z 610.687,A -85,B 0,C 180,E1 -6565.042,E2 -6565.042} C_VEL
LIN {X 0,Y 487.941,Z 613.187,A -85,B 0,C 180,E1 -6566.697,E2 -6566.697} C_VEL
LIN {X 0,Y 487.885,Z 614.595,A -85,B 0,C 180,E1 -6568.349,E2 -6568.349} C_VEL
LIN {X 0,Y 487.814,Z 615.128,A -85,B 0,C 180,E1 -6570,E2 -6570} C_VEL
LIN {X 0,Y 487.885,Z 614.603,A -85,B 0,C 180,E1 -6571.651,E2 -6571.651} C_VEL
LIN {X 0,Y 487.941,Z 613.201,A -85,B 0,C 180,E1 -6573.303,E2 -6573.303} C_VEL
LIN {X 0,Y 487.907,Z 610.712,A -85,B 0,C 180,E1 -6574.958,E2 -6574.958} C_VEL
LIN {X 0,Y 487.995,Z 607.29,A -85,B 0,C 180,E1 -6576.616,E2 -6576.616} C_VEL
LIN {X 0,Y 488.09,Z 601.431,A -85,B 0,C 180,E1 -6578.696,E2 -6578.696} C_VEL
LIN {X 0,Y 488.383,Z 593.725,A -85,B 0,C 180,E1 -6580.782,E2 -6580.782} C_VEL
LIN {X 0,Y 488.775,Z 585.031,A -85,B 0,C 180,E1 -6582.667,E2 -6582.667} C_VEL
LIN {X 0,Y 489.171,Z 575.64,A -85,B 0,C 180,E1 -6584.349,E2 -6584.349} C_VEL
LIN {X 0,Y 489.758,Z 565.976,A -85,B 0,C 180,E1 -6585.822,E2 -6585.822} C_VEL
LIN {X 0,Y 490.478,Z 554.714,A -85,B 0,C 180,E1 -6587.297,E2 -6587.297} C_VEL
LIN {X 0,Y 491.289,Z 542.454,A -85,B 0,C 180,E1 -6588.668,E2 -6588.668} C_VEL
LIN {X 0,Y 492.186,Z 529.059,A -85,B 0,C 180,E1 -6589.931,E2 -6589.931} C_VEL
LIN {X 0,Y 493.079,Z 515.868,A -85,B 0,C 180,E1 -6590.984,E2 -6590.984} C_VEL
LIN {X 0,Y 493.897,Z 502.577,A -85,B 0,C 180,E1 -6591.891,E2 -6591.891} C_VEL
LIN {X 0,Y 494.855,Z 486.828,A -85,B 0,C 180,E1 -6592.768,E2 -6592.768} C_VEL
LIN {X 0,Y 495.539,Z 472.737,A -85,B 0,C 180,E1 -6593.398,E2 -6593.398} C_VEL
LIN {X 0,Y 496.167,Z 457.071,A -85,B 0,C 180,E1 -6593.948,E2 -6593.948} C_VEL
LIN {X 0,Y 496.644,Z 441.725,A -85,B 0,C 180,E1 -6594.338,E2 -6594.338} C_VEL
LIN {X 0,Y 497.235,Z 401.874,A -85,B 0,C 180,E1 -6594.964,E2 -6594.964} C_VEL
LIN {X 0,Y 498.885,Z 253.751,A -85,B 0,C 180,E1 -6597.219,E2 -6597.219} C_VEL
LIN {X 0,Y 495.152,Z 232.833,A -85,B 0,C 180,E1 -6597.79,E2 -6597.79} C_VEL
LIN {X 0,Y 495.818,Z 220.711,A -85,B 0,C 180,E1 -6599.011,E2 -6599.011} C_VEL
LIN {X 0,Y 490.844,Z 203.842,A -85,B 0,C 180,E1 -6601.116,E2 -6601.116} C_VEL
LIN {X 0,Y 488.716,Z 196.911,A -85,B 0,C 180,E1 -6602.046,E2 -6602.046} C_VEL
LIN {X 0,Y 488.713,Z 196.922,A -85,B 0,C 180,E1 -6605.115,E2 -6605.115} C_VEL
LIN {X 0,Y 488.674,Z 196.925,A -85,B 0,C 180,E1 -6608.2,E2 -6608.2} C_VEL
LIN {X 0,Y 488.716,Z 196.916,A -85,B 0,C 180,E1 -6610.345,E2 -6610.345} C_VEL
LIN {X 0,Y 488.675,Z 196.925,A -85,B 0,C 180,E1 -6613.655,E2 -6613.655} C_VEL
LIN {X 0,Y 488.673,Z 196.92,A -85,B 0,C 180,E1 -6616.344,E2 -6616.344} C_VEL
LIN {X 0,Y 488.7,Z 196.917,A -85,B 0,C 180,E1 -6619.673,E2 -6619.673} C_VEL
LIN {X 0,Y 488.676,Z 196.923,A -85,B 0,C 180,E1 -6622.841,E2 -6622.841} C_VEL
LIN {X 0,Y 488.72,Z 196.917,A -85,B 0,C 180,E1 -6625.887,E2 -6625.887} C_VEL
LIN {X 0,Y 488.689,Z 196.919,A -85,B 0,C 180,E1 -6628.82,E2 -6628.82} C_VEL
LIN {X 0,Y 488.739,Z 196.915,A -85,B 0,C 180,E1 -6631.671,E2 -6631.671} C_VEL
LIN {X 0,Y 488.749,Z 196.905,A -85,B 0,C 180,E1 -6633.528,E2 -6633.528} C_VEL
LIN {X 0,Y 488.672,Z 196.923,A -85,B 0,C 180,E1 -6636.254,E2 -6636.254} C_VEL
LIN {X 0,Y 488.743,Z 196.909,A -85,B 0,C 180,E1 -6639.176,E2 -6639.176} C_VEL
LIN {X 0,Y 488.744,Z 196.905,A -85,B 0,C 180,E1 -6641.632,E2 -6641.632} C_VEL
LIN {X 0,Y 488.758,Z 196.913,A -85,B 0,C 180,E1 -6645,E2 -6645} C_VEL
LIN {X 0,Y 488.802,Z 196.897,A -85,B 0,C 180,E1 -6648.388,E2 -6648.388} C_VEL
LIN {X 0,Y 488.782,Z 196.908,A -85,B 0,C 180,E1 -6651.733,E2 -6651.733} C_VEL
LIN {X 0,Y 488.842,Z 196.905,A -85,B 0,C 180,E1 -6654.224,E2 -6654.224} C_VEL
LIN {X 0,Y 488.955,Z 196.87,A -85,B 0,C 180,E1 -6657.529,E2 -6657.529} C_VEL
LIN {X 0,Y 488.951,Z 196.889,A -85,B 0,C 180,E1 -6660.824,E2 -6660.824} C_VEL
LIN {X 0,Y 488.956,Z 196.89,A -85,B 0,C 180,E1 -6662.471,E2 -6662.471} C_VEL
LIN {X 0,Y 488.85,Z 196.893,A -85,B 0,C 180,E1 -6665.776,E2 -6665.776} C_VEL
LIN {X 0,Y 488.813,Z 196.911,A -85,B 0,C 180,E1 -6668.266,E2 -6668.266} C_VEL
LIN {X 0,Y 488.802,Z 196.902,A -85,B 0,C 180,E1 -6671.612,E2 -6671.612} C_VEL
LIN {X 0,Y 488.759,Z 196.911,A -85,B 0,C 180,E1 -6675,E2 -6675} C_VEL
LIN {X 0,Y 488.752,Z 196.905,A -85,B 0,C 180,E1 -6678.442,E2 -6678.442} C_VEL
LIN {X 0,Y 488.704,Z 196.917,A -85,B 0,C 180,E1 -6681.071,E2 -6681.071} C_VEL
LIN {X 0,Y 488.691,Z 196.924,A -85,B 0,C 180,E1 -6683.745,E2 -6683.745} C_VEL
LIN {X 0,Y 488.789,Z 196.904,A -85,B 0,C 180,E1 -6686.944,E2 -6686.944} C_VEL
LIN {X 0,Y 488.716,Z 196.915,A -85,B 0,C 180,E1 -6690.365,E2 -6690.365} C_VEL
LIN {X 0,Y 488.733,Z 196.914,A -85,B 0,C 180,E1 -6693.485,E2 -6693.485} C_VEL
LIN {X 0,Y 488.686,Z 196.919,A -85,B 0,C 180,E1 -6696.356,E2 -6696.356} C_VEL
LIN {X 0,Y 488.698,Z 196.917,A -85,B 0,C 180,E1 -6699.254,E2 -6699.254} C_VEL
LIN {X 0,Y 488.706,Z 196.925,A -85,B 0,C 180,E1 -6701.6,E2 -6701.6} C_VEL
LIN {X 0,Y 488.699,Z 196.916,A -85,B 0,C 180,E1 -6704.803,E2 -6704.803} C_VEL
LIN {X 0,Y 488.69,Z 196.925,A -85,B 0,C 180,E1 -6707.475,E2 -6707.475} C_VEL
LIN {X 0,Y 488.731,Z 196.918,A -85,B 0,C 180,E1 -6709.677,E2 -6709.677} C_VEL
LIN {X 0,Y 488.677,Z 196.923,A -85,B 0,C 180,E1 -6712.841,E2 -6712.841} C_VEL
LIN {X 0,Y 488.73,Z 196.918,A -85,B 0,C 180,E1 -6715.887,E2 -6715.887} C_VEL
LIN {X 0,Y 488.691,Z 196.918,A -85,B 0,C 180,E1 -6718.82,E2 -6718.82} C_VEL
LIN {X 0,Y 488.743,Z 196.914,A -85,B 0,C 180,E1 -6721.671,E2 -6721.671} C_VEL
LIN {X 0,Y 488.742,Z 196.914,A -85,B 0,C 180,E1 -6724.35,E2 -6724.35} C_VEL
LIN {X 0,Y 488.097,Z 197.001,A -85,B 0,C 180,E1 -6725.038,E2 -6725.038} C_VEL
LIN {X 0,Y 485.228,Z 197.356,A -85,B 0,C 180,E1 -6726.155,E2 -6726.155} C_VEL
LIN {X 0,Y 482.781,Z 197.66,A -85,B 0,C 180,E1 -6727.054,E2 -6727.054} C_VEL
LIN {X 0,Y 481.723,Z 197.791,A -85,B 0,C 180,E1 -6727.75,E2 -6727.75} C_VEL
LIN {X 0,Y 481.634,Z 197.801,A -85,B 0,C 180,E1 -6727.985,E2 -6727.985} C_VEL
LIN {X 0,Y 481.704,Z 197.784,A -85,B 0,C 180,E1 -6730.393,E2 -6730.393} C_VEL
LIN {X 0,Y 481.678,Z 197.798,A -85,B 0,C 180,E1 -6733.033,E2 -6733.033} C_VEL
LIN {X 0,Y 481.689,Z 197.783,A -85,B 0,C 180,E1 -6735.639,E2 -6735.639} C_VEL
LIN {X 0,Y 481.751,Z 197.787,A -85,B 0,C 180,E1 -6738.215,E2 -6738.215} C_VEL
LIN {X 0,Y 481.763,Z 197.787,A -85,B 0,C 180,E1 -6741.612,E2 -6741.612} C_VEL
LIN {X 0,Y 481.777,Z 197.789,A -85,B 0,C 180,E1 -6744.979,E2 -6744.979} C_VEL
LIN {X 0,Y 481.675,Z 197.812,A -85,B 0,C 180,E1 -6746.157,E2 -6746.157} C_VEL
LIN {X 0,Y 484.922,Z 208.393,A -85,B 0,C 180,E1 -6747.654,E2 -6747.654} C_VEL
LIN {X 0,Y 492.297,Z 224.861,A -85,B 0,C 180,E1 -6748.385,E2 -6748.385} C_VEL
LIN {X 0,Y 492.836,Z 228.233,A -85,B 0,C 180,E1 -6748.473,E2 -6748.473} C_VEL
LIN {X 0,Y 490.363,Z 414.563,A -85,B 0,C 180,E1 -6751.36,E2 -6751.36} C_VEL
LIN {X 0,Y 489.894,Z 431.455,A -85,B 0,C 180,E1 -6751.798,E2 -6751.798} C_VEL
LIN {X 0,Y 489.173,Z 447.243,A -85,B 0,C 180,E1 -6752.367,E2 -6752.367} C_VEL
LIN {X 0,Y 488.413,Z 462.69,A -85,B 0,C 180,E1 -6753.093,E2 -6753.093} C_VEL
LIN {X 0,Y 487.575,Z 477.063,A -85,B 0,C 180,E1 -6753.926,E2 -6753.926} C_VEL
LIN {X 0,Y 486.597,Z 491.815,A -85,B 0,C 180,E1 -6754.971,E2 -6754.971} C_VEL
LIN {X 0,Y 485.661,Z 505.381,A -85,B 0,C 180,E1 -6756.126,E2 -6756.126} C_VEL
LIN {X 0,Y 484.75,Z 517.085,A -85,B 0,C 180,E1 -6757.288,E2 -6757.288} C_VEL
LIN {X 0,Y 483.852,Z 529.384,A -85,B 0,C 180,E1 -6758.717,E2 -6758.717} C_VEL
LIN {X 0,Y 483.022,Z 540.654,A -85,B 0,C 180,E1 -6760.267,E2 -6760.267} C_VEL
LIN {X 0,Y 482.423,Z 549.918,A -85,B 0,C 180,E1 -6761.768,E2 -6761.768} C_VEL
LIN {X 0,Y 481.818,Z 559.012,A -85,B 0,C 180,E1 -6763.496,E2 -6763.496} C_VEL
LIN {X 0,Y 481.409,Z 566.657,A -85,B 0,C 180,E1 -6765.235,E2 -6765.235} C_VEL
LIN {X 0,Y 481.141,Z 572.925,A -85,B 0,C 180,E1 -6766.986,E2 -6766.986} C_VEL
LIN {X 0,Y 480.979,Z 578.003,A -85,B 0,C 180,E1 -6768.751,E2 -6768.751} C_VEL
LIN {X 0,Y 480.81,Z 582.27,A -85,B 0,C 180,E1 -6770.694,E2 -6770.694} C_VEL
LIN {X 0,Y 480.72,Z 584.8,A -85,B 0,C 180,E1 -6772.34,E2 -6772.34} C_VEL
LIN {X 0,Y 480.643,Z 586.526,A -85,B 0,C 180,E1 -6774.168,E2 -6774.168} C_VEL
LIN {X 0,Y 480.668,Z 587.163,A -85,B 0,C 180,E1 -6776.016,E2 -6776.016} C_VEL
LIN {X 0,Y 480.685,Z 586.553,A -85,B 0,C 180,E1 -6777.895,E2 -6777.895} C_VEL
LIN {X 0,Y 480.742,Z 584.752,A -85,B 0,C 180,E1 -6779.804,E2 -6779.804} C_VEL
LIN {X 0,Y 480.887,Z 581.655,A -85,B 0,C 180,E1 -6781.743,E2 -6781.743} C_VEL
LIN {X 0,Y 481.021,Z 577.085,A -85,B 0,C 180,E1 -6783.724,E2 -6783.724} C_VEL
LIN {X 0,Y 481.226,Z 571.994,A -85,B 0,C 180,E1 -6785.399,E2 -6785.399} C_VEL
LIN {X 0,Y 481.524,Z 564.969,A -85,B 0,C 180,E1 -6787.279,E2 -6787.279} C_VEL
LIN {X 0,Y 481.926,Z 557.969,A -85,B 0,C 180,E1 -6788.834,E2 -6788.834} C_VEL
LIN {X 0,Y 482.502,Z 548.476,A -85,B 0,C 180,E1 -6790.593,E2 -6790.593} C_VEL
LIN {X 0,Y 483.195,Z 538.741,A -85,B 0,C 180,E1 -6792.116,E2 -6792.116} C_VEL
LIN {X 0,Y 483.907,Z 528.324,A -85,B 0,C 180,E1 -6793.524,E2 -6793.524} C_VEL
LIN {X 0,Y 484.845,Z 516.309,A -85,B 0,C 180,E1 -6794.905,E2 -6794.905} C_VEL
LIN {X 0,Y 485.866,Z 502.872,A -85,B 0,C 180,E1 -6796.21,E2 -6796.21} C_VEL
LIN {X 0,Y 486.771,Z 490.039,A -85,B 0,C 180,E1 -6797.267,E2 -6797.267} C_VEL
LIN {X 0,Y 487.641,Z 476.29,A -85,B 0,C 180,E1 -6798.229,E2 -6798.229} C_VEL
LIN {X 0,Y 488.651,Z 460.235,A -85,B 0,C 180,E1 -6799.141,E2 -6799.141} C_VEL
LIN {X 0,Y 489.34,Z 445.005,A -85,B 0,C 180,E1 -6799.827,E2 -6799.827} C_VEL
LIN {X 0,Y 489.987,Z 428.76,A -85,B 0,C 180,E1 -6800.384,E2 -6800.384} C_VEL
LIN {X 0,Y 490.456,Z 412.597,A -85,B 0,C 180,E1 -6800.774,E2 -6800.774} C_VEL
LIN {X 0,Y 492.879,Z 227.39,A -85,B 0,C 180,E1 -6803.655,E2 -6803.655} C_VEL
LIN {X 0,Y 491.973,Z 224.001,A -85,B 0,C 180,E1 -6803.768,E2 -6803.768} C_VEL
LIN {X 0,Y 484.904,Z 208.594,A -85,B 0,C 180,E1 -6804.503,E2 -6804.503} C_VEL
LIN {X 0,Y 481.686,Z 197.796,A -85,B 0,C 180,E1 -6806.068,E2 -6806.068} C_VEL
LIN {X 0,Y 481.641,Z 197.804,A -85,B 0,C 180,E1 -6809.418,E2 -6809.418} C_VEL
LIN {X 0,Y 481.653,Z 197.801,A -85,B 0,C 180,E1 -6812.165,E2 -6812.165} C_VEL
LIN {X 0,Y 481.666,Z 197.799,A -85,B 0,C 180,E1 -6814.967,E2 -6814.967} C_VEL
LIN {X 0,Y 481.64,Z 197.796,A -85,B 0,C 180,E1 -6817.704,E2 -6817.704} C_VEL
LIN {X 0,Y 481.696,Z 197.796,A -85,B 0,C 180,E1 -6820.393,E2 -6820.393} C_VEL
LIN {X 0,Y 481.671,Z 197.798,A -85,B 0,C 180,E1 -6823.033,E2 -6823.033} C_VEL
LIN {X 0,Y 481.681,Z 197.795,A -85,B 0,C 180,E1 -6825.639,E2 -6825.639} C_VEL
LIN {X 0,Y 481.743,Z 197.783,A -85,B 0,C 180,E1 -6828.215,E2 -6828.215} C_VEL
LIN {X 0,Y 481.733,Z 197.787,A -85,B 0,C 180,E1 -6831.611,E2 -6831.611} C_VEL
LIN {X 0,Y 481.799,Z 197.782,A -85,B 0,C 180,E1 -6834.139,E2 -6834.139} C_VEL
LIN {X 0,Y 481.919,Z 197.764,A -85,B 0,C 180,E1 -6837.493,E2 -6837.493} C_VEL
LIN {X 0,Y 481.899,Z 197.768,A -85,B 0,C 180,E1 -6840.836,E2 -6840.836} C_VEL
LIN {X 0,Y 481.92,Z 197.766,A -85,B 0,C 180,E1 -6842.507,E2 -6842.507} C_VEL
LIN {X 0,Y 481.808,Z 197.781,A -85,B 0,C 180,E1 -6845.86,E2 -6845.86} C_VEL
LIN {X 0,Y 481.756,Z 197.788,A -85,B 0,C 180,E1 -6848.388,E2 -6848.388} C_VEL
LIN {X 0,Y 481.744,Z 197.788,A -85,B 0,C 180,E1 -6851.785,E2 -6851.785} C_VEL
LIN {X 0,Y 481.736,Z 197.788,A -85,B 0,C 180,E1 -6855.224,E2 -6855.224} C_VEL
LIN {X 0,Y 481.706,Z 197.789,A -85,B 0,C 180,E1 -6858.722,E2 -6858.722} C_VEL
LIN {X 0,Y 481.64,Z 197.802,A -85,B 0,C 180,E1 -6861.395,E2 -6861.395} C_VEL
LIN {X 0,Y 481.671,Z 197.797,A -85,B 0,C 180,E1 -6864.113,E2 -6864.113} C_VEL
LIN {X 0,Y 481.746,Z 197.786,A -85,B 0,C 180,E1 -6867.141,E2 -6867.141} C_VEL
LIN {X 0,Y 481.673,Z 197.802,A -85,B 0,C 180,E1 -6869.741,E2 -6869.741} C_VEL
LIN {X 0,Y 481.667,Z 197.798,A -85,B 0,C 180,E1 -6872.674,E2 -6872.674} C_VEL
LIN {X 0,Y 481.632,Z 197.806,A -85,B 0,C 180,E1 -6875.71,E2 -6875.71} C_VEL
LIN {X 0,Y 481.665,Z 197.801,A -85,B 0,C 180,E1 -6878.859,E2 -6878.859} C_VEL
LIN {X 0,Y 481.647,Z 197.802,A -85,B 0,C 180,E1 -6881.913,E2 -6881.913} C_VEL
LIN {X 0,Y 481.654,Z 197.802,A -85,B 0,C 180,E1 -6884.458,E2 -6884.458} C_VEL
LIN {X 0,Y 481.642,Z 197.803,A -85,B 0,C 180,E1 -6887.84,E2 -6887.84} C_VEL
LIN {X 0,Y 481.676,Z 197.799,A -85,B 0,C 180,E1 -6890.652,E2 -6890.652} C_VEL
LIN {X 0,Y 481.623,Z 197.807,A -85,B 0,C 180,E1 -6893.377,E2 -6893.377} C_VEL
LIN {X 0,Y 481.706,Z 197.791,A -85,B 0,C 180,E1 -6896.331,E2 -6896.331} C_VEL
LIN {X 0,Y 481.683,Z 197.934,A -85,B 0,C 180,E1 -6897.591,E2 -6897.591} C_VEL
LIN {X 0,Y 487.196,Z 215.802,A -85,B 0,C 180,E1 -6899.942,E2 -6899.942} C_VEL
LIN {X 0,Y 489.023,Z 222.221,A -85,B 0,C 180,E1 -6900.75,E2 -6900.75} C_VEL
LIN {X 0,Y 488.594,Z 232.459,A -85,B 0,C 180,E1 -6901.798,E2 -6901.798} C_VEL
LIN {X 0,Y 492.662,Z 255.793,A -85,B 0,C 180,E1 -6902.437,E2 -6902.437} C_VEL
LIN {X 0,Y 490.258,Z 438.881,A -85,B 0,C 180,E1 -6905.276,E2 -6905.276} C_VEL
LIN {X 0,Y 489.669,Z 454.711,A -85,B 0,C 180,E1 -6905.658,E2 -6905.658} C_VEL
LIN {X 0,Y 489.037,Z 470.921,A -85,B 0,C 180,E1 -6906.217,E2 -6906.217} C_VEL
LIN {X 0,Y 488.198,Z 486.34,A -85,B 0,C 180,E1 -6906.904,E2 -6906.904} C_VEL
LIN {X 0,Y 487.246,Z 502.387,A -85,B 0,C 180,E1 -6907.813,E2 -6907.813} C_VEL
LIN {X 0,Y 486.258,Z 516.85,A -85,B 0,C 180,E1 -6908.819,E2 -6908.819} C_VEL
LIN {X 0,Y 485.369,Z 529.792,A -85,B 0,C 180,E1 -6909.887,E2 -6909.887} C_VEL
LIN {X 0,Y 484.336,Z 543.028,A -85,B 0,C 180,E1 -6911.165,E2 -6911.165} C_VEL
LIN {X 0,Y 483.562,Z 554.33,A -85,B 0,C 180,E1 -6912.448,E2 -6912.448} C_VEL
LIN {X 0,Y 482.768,Z 565.616,A -85,B 0,C 180,E1 -6913.943,E2 -6913.943} C_VEL
LIN {X 0,Y 482.206,Z 575.306,A -85,B 0,C 180,E1 -6915.439,E2 -6915.439} C_VEL
LIN {X 0,Y 481.719,Z 584.72,A -85,B 0,C 180,E1 -6917.145,E2 -6917.145} C_VEL
LIN {X 0,Y 481.306,Z 593.437,A -85,B 0,C 180,E1 -6919.058,E2 -6919.058} C_VEL
LIN {X 0,Y 481.023,Z 601.163,A -85,B 0,C 180,E1 -6921.176,E2 -6921.176} C_VEL
LIN {X 0,Y 480.903,Z 607.04,A -85,B 0,C 180,E1 -6923.286,E2 -6923.286} C_VEL
LIN {X 0,Y 480.832,Z 610.478,A -85,B 0,C 180,E1 -6924.969,E2 -6924.969} C_VEL
LIN {X 0,Y 480.846,Z 612.979,A -85,B 0,C 180,E1 -6926.649,E2 -6926.649} C_VEL
LIN {X 0,Y 480.816,Z 614.39,A -85,B 0,C 180,E1 -6928.325,E2 -6928.325} C_VEL
LIN {X 0,Y 480.738,Z 614.924,A -85,B 0,C 180,E1 -6930,E2 -6930} C_VEL
LIN {X 0,Y 480.816,Z 614.399,A -85,B 0,C 180,E1 -6931.675,E2 -6931.675} C_VEL
LIN {X 0,Y 480.846,Z 612.997,A -85,B 0,C 180,E1 -6933.352,E2 -6933.352} C_VEL
LIN {X 0,Y 480.832,Z 610.508,A -85,B 0,C 180,E1 -6935.031,E2 -6935.031} C_VEL
LIN {X 0,Y 480.904,Z 607.083,A -85,B 0,C 180,E1 -6936.714,E2 -6936.714} C_VEL
LIN {X 0,Y 481.029,Z 601.223,A -85,B 0,C 180,E1 -6938.825,E2 -6938.825} C_VEL
LIN {X 0,Y 481.315,Z 593.513,A -85,B 0,C 180,E1 -6940.942,E2 -6940.942} C_VEL
LIN {X 0,Y 481.721,Z 584.816,A -85,B 0,C 180,E1 -6942.855,E2 -6942.855} C_VEL
LIN {X 0,Y 482.21,Z 575.423,A -85,B 0,C 180,E1 -6944.561,E2 -6944.561} C_VEL
LIN {X 0,Y 482.876,Z 565.163,A -85,B 0,C 180,E1 -6946.139,E2 -6946.139} C_VEL
LIN {X 0,Y 483.592,Z 554.482,A -85,B 0,C 180,E1 -6947.551,E2 -6947.551} C_VEL
LIN {X 0,Y 484.454,Z 542.214,A -85,B 0,C 180,E1 -6948.941,E2 -6948.941} C_VEL
LIN {X 0,Y 485.408,Z 528.911,A -85,B 0,C 180,E1 -6950.212,E2 -6950.212} C_VEL
LIN {X 0,Y 486.374,Z 515.612,A -85,B 0,C 180,E1 -6951.288,E2 -6951.288} C_VEL
LIN {X 0,Y 487.344,Z 501.22,A -85,B 0,C 180,E1 -6952.269,E2 -6952.269} C_VEL
LIN {X 0,Y 488.266,Z 486.541,A -85,B 0,C 180,E1 -6953.093,E2 -6953.093} C_VEL
LIN {X 0,Y 489.056,Z 471.113,A -85,B 0,C 180,E1 -6953.783,E2 -6953.783} C_VEL
LIN {X 0,Y 489.701,Z 454.858,A -85,B 0,C 180,E1 -6954.341,E2 -6954.341} C_VEL
LIN {X 0,Y 490.264,Z 438.827,A -85,B 0,C 180,E1 -6954.726,E2 -6954.726} C_VEL
LIN {X 0,Y 492.628,Z 255.65,A -85,B 0,C 180,E1 -6957.557,E2 -6957.557} C_VEL
LIN {X 0,Y 488.612,Z 232.754,A -85,B 0,C 180,E1 -6958.18,E2 -6958.18} C_VEL
LIN {X 0,Y 489.061,Z 222.391,A -85,B 0,C 180,E1 -6959.248,E2 -6959.248} C_VEL
LIN {X 0,Y 483.705,Z 204.402,A -85,B 0,C 180,E1 -6961.538,E2 -6961.538} C_VEL
LIN {X 0,Y 481.67,Z 197.784,A -85,B 0,C 180,E1 -6962.429,E2 -6962.429} C_VEL
LIN {X 0,Y 481.658,Z 197.8,A -85,B 0,C 180,E1 -6965.204,E2 -6965.204} C_VEL
LIN {X 0,Y 481.668,Z 197.802,A -85,B 0,C 180,E1 -6968.859,E2 -6968.859} C_VEL
LIN {X 0,Y 481.643,Z 197.799,A -85,B 0,C 180,E1 -6971.912,E2 -6971.912} C_VEL
LIN {X 0,Y 481.651,Z 197.8,A -85,B 0,C 180,E1 -6974.458,E2 -6974.458} C_VEL
LIN {X 0,Y 481.64,Z 197.8,A -85,B 0,C 180,E1 -6977.839,E2 -6977.839} C_VEL
LIN {X 0,Y 481.654,Z 197.799,A -85,B 0,C 180,E1 -6980.655,E2 -6980.655} C_VEL
LIN {X 0,Y 481.624,Z 197.796,A -85,B 0,C 180,E1 -6983.376,E2 -6983.376} C_VEL
LIN {X 0,Y 481.673,Z 197.797,A -85,B 0,C 180,E1 -6986.327,E2 -6986.327} C_VEL
LIN {X 0,Y 481.647,Z 197.797,A -85,B 0,C 180,E1 -6989.417,E2 -6989.417} C_VEL
LIN {X 0,Y 481.695,Z 197.794,A -85,B 0,C 180,E1 -6992.168,E2 -6992.168} C_VEL
LIN {X 0,Y 481.689,Z 197.792,A -85,B 0,C 180,E1 -6994.968,E2 -6994.968} C_VEL
LIN {X 0,Y 481.644,Z 197.799,A -85,B 0,C 180,E1 -6997.705,E2 -6997.705} C_VEL
LIN {X 0,Y 481.699,Z 197.785,A -85,B 0,C 180,E1 -7000.393,E2 -7000.393} C_VEL
LIN {X 0,Y 481.672,Z 197.796,A -85,B 0,C 180,E1 -7003.033,E2 -7003.033} C_VEL
LIN {X 0,Y 481.685,Z 197.792,A -85,B 0,C 180,E1 -7005.639,E2 -7005.639} C_VEL
LIN {X 0,Y 481.747,Z 197.774,A -85,B 0,C 180,E1 -7008.215,E2 -7008.215} C_VEL
LIN {X 0,Y 481.737,Z 197.785,A -85,B 0,C 180,E1 -7011.611,E2 -7011.611} C_VEL
LIN {X 0,Y 481.803,Z 197.783,A -85,B 0,C 180,E1 -7014.139,E2 -7014.139} C_VEL
LIN {X 0,Y 481.922,Z 197.745,A -85,B 0,C 180,E1 -7017.493,E2 -7017.493} C_VEL
LIN {X 0,Y 481.902,Z 197.767,A -85,B 0,C 180,E1 -7020.836,E2 -7020.836} C_VEL
LIN {X 0,Y 481.923,Z 197.766,A -85,B 0,C 180,E1 -7022.507,E2 -7022.507} C_VEL
LIN {X 0,Y 481.811,Z 197.77,A -85,B 0,C 180,E1 -7025.86,E2 -7025.86} C_VEL
LIN {X 0,Y 481.758,Z 197.788,A -85,B 0,C 180,E1 -7028.388,E2 -7028.388} C_VEL
LIN {X 0,Y 481.747,Z 197.781,A -85,B 0,C 180,E1 -7031.785,E2 -7031.785} C_VEL
LIN {X 0,Y 481.74,Z 197.785,A -85,B 0,C 180,E1 -7035.224,E2 -7035.224} C_VEL
LIN {X 0,Y 481.709,Z 197.78,A -85,B 0,C 180,E1 -7038.722,E2 -7038.722} C_VEL
LIN {X 0,Y 481.643,Z 197.798,A -85,B 0,C 180,E1 -7041.395,E2 -7041.395} C_VEL
LIN {X 0,Y 481.674,Z 197.792,A -85,B 0,C 180,E1 -7044.113,E2 -7044.113} C_VEL
LIN {X 0,Y 481.744,Z 197.782,A -85,B 0,C 180,E1 -7047.139,E2 -7047.139} C_VEL
LIN {X 0,Y 481.685,Z 197.799,A -85,B 0,C 180,E1 -7049.741,E2 -7049.741} C_VEL
LIN {X 0,Y 481.67,Z 197.789,A -85,B 0,C 180,E1 -7052.674,E2 -7052.674} C_VEL
LIN {X 0,Y 481.64,Z 197.804,A -85,B 0,C 180,E1 -7055.709,E2 -7055.709} C_VEL
LIN {X 0,Y 481.668,Z 197.789,A -85,B 0,C 180,E1 -7058.859,E2 -7058.859} C_VEL
LIN {X 0,Y 481.651,Z 197.799,A -85,B 0,C 180,E1 -7061.913,E2 -7061.913} C_VEL
LIN {X 0,Y 481.652,Z 197.793,A -85,B 0,C 180,E1 -7064.458,E2 -7064.458} C_VEL
LIN {X 0,Y 481.645,Z 197.797,A -85,B 0,C 180,E1 -7067.839,E2 -7067.839} C_VEL
LIN {X 0,Y 481.659,Z 197.796,A -85,B 0,C 180,E1 -7070.654,E2 -7070.654} C_VEL
LIN {X 0,Y 481.626,Z 197.8,A -85,B 0,C 180,E1 -7073.376,E2 -7073.376} C_VEL
LIN {X 0,Y 481.708,Z 197.791,A -85,B 0,C 180,E1 -7076.33,E2 -7076.33} C_VEL
LIN {X 0,Y 481.65,Z 197.801,A -85,B 0,C 180,E1 -7079.417,E2 -7079.417} C_VEL
LIN {X 0,Y 481.699,Z 197.789,A -85,B 0,C 180,E1 -7082.168,E2 -7082.168} C_VEL
LIN {X 0,Y 481.717,Z 197.795,A -85,B 0,C 180,E1 -7084.97,E2 -7084.97} C_VEL
LIN {X 0,Y 481.634,Z 197.801,A -85,B 0,C 180,E1 -7087.985,E2 -7087.985} C_VEL
LIN {X 0,Y 480.968,Z 197.888,A -85,B 0,C 180,E1 -7088.683,E2 -7088.683} C_VEL
LIN {X 0,Y 478.141,Z 198.228,A -85,B 0,C 180,E1 -7089.818,E2 -7089.818} C_VEL
LIN {X 0,Y 475.755,Z 198.522,A -85,B 0,C 180,E1 -7090.732,E2 -7090.732} C_VEL
LIN {X 0,Y 474.73,Z 198.65,A -85,B 0,C 180,E1 -7091.438,E2 -7091.438} C_VEL
LIN {X 0,Y 474.646,Z 198.663,A -85,B 0,C 180,E1 -7091.677,E2 -7091.677} C_VEL
LIN {X 0,Y 474.699,Z 198.668,A -85,B 0,C 180,E1 -7094.544,E2 -7094.544} C_VEL
LIN {X 0,Y 474.704,Z 198.665,A -85,B 0,C 180,E1 -7098.037,E2 -7098.037} C_VEL
LIN {X 0,Y 474.728,Z 198.665,A -85,B 0,C 180,E1 -7101.486,E2 -7101.486} C_VEL
LIN {X 0,Y 474.748,Z 198.665,A -85,B 0,C 180,E1 -7104.904,E2 -7104.904} C_VEL
LIN {X 0,Y 474.641,Z 198.857,A -85,B 0,C 180,E1 -7105.781,E2 -7105.781} C_VEL
LIN {X 0,Y 477.832,Z 208.793,A -85,B 0,C 180,E1 -7107.203,E2 -7107.203} C_VEL
LIN {X 0,Y 486.283,Z 227.411,A -85,B 0,C 180,E1 -7108.057,E2 -7108.057} C_VEL
LIN {X 0,Y 486.528,Z 231.315,A -85,B 0,C 180,E1 -7108.137,E2 -7108.137} C_VEL
LIN {X 0,Y 483.917,Z 414.693,A -85,B 0,C 180,E1 -7111.014,E2 -7111.014} C_VEL
LIN {X 0,Y 483.402,Z 431.652,A -85,B 0,C 180,E1 -7111.458,E2 -7111.458} C_VEL
LIN {X 0,Y 482.651,Z 447.443,A -85,B 0,C 180,E1 -7112.034,E2 -7112.034} C_VEL
LIN {X 0,Y 481.791,Z 463.865,A -85,B 0,C 180,E1 -7112.822,E2 -7112.822} C_VEL
LIN {X 0,Y 480.778,Z 479.617,A -85,B 0,C 180,E1 -7113.771,E2 -7113.771} C_VEL
LIN {X 0,Y 479.809,Z 493.527,A -85,B 0,C 180,E1 -7114.788,E2 -7114.788} C_VEL
LIN {X 0,Y 478.786,Z 507.347,A -85,B 0,C 180,E1 -7116.003,E2 -7116.003} C_VEL
LIN {X 0,Y 477.846,Z 518.762,A -85,B 0,C 180,E1 -7117.181,E2 -7117.181} C_VEL
LIN {X 0,Y 476.902,Z 530.783,A -85,B 0,C 180,E1 -7118.624,E2 -7118.624} C_VEL
LIN {X 0,Y 476.043,Z 541.964,A -85,B 0,C 180,E1 -7120.204,E2 -7120.204} C_VEL
LIN {X 0,Y 475.324,Z 552.315,A -85,B 0,C 180,E1 -7121.946,E2 -7121.946} C_VEL
LIN {X 0,Y 474.733,Z 561.018,A -85,B 0,C 180,E1 -7123.701,E2 -7123.701} C_VEL
LIN {X 0,Y 474.273,Z 568.782,A -85,B 0,C 180,E1 -7125.593,E2 -7125.593} C_VEL
LIN {X 0,Y 474.046,Z 574.371,A -85,B 0,C 180,E1 -7127.248,E2 -7127.248} C_VEL
LIN {X 0,Y 473.877,Z 579.19,A -85,B 0,C 180,E1 -7129.043,E2 -7129.043} C_VEL
LIN {X 0,Y 473.717,Z 582.882,A -85,B 0,C 180,E1 -7130.858,E2 -7130.858} C_VEL
LIN {X 0,Y 473.599,Z 585.517,A -85,B 0,C 180,E1 -7132.695,E2 -7132.695} C_VEL
LIN {X 0,Y 473.555,Z 586.961,A -85,B 0,C 180,E1 -7134.553,E2 -7134.553} C_VEL
LIN {X 0,Y 473.587,Z 587.303,A -85,B 0,C 180,E1 -7136.435,E2 -7136.435} C_VEL
LIN {X 0,Y 473.622,Z 586.509,A -85,B 0,C 180,E1 -7138.348,E2 -7138.348} C_VEL
LIN {X 0,Y 473.707,Z 584.393,A -85,B 0,C 180,E1 -7140.293,E2 -7140.293} C_VEL
LIN {X 0,Y 473.821,Z 580.929,A -85,B 0,C 180,E1 -7142.279,E2 -7142.279} C_VEL
LIN {X 0,Y 474.015,Z 576.014,A -85,B 0,C 180,E1 -7144.291,E2 -7144.291} C_VEL
LIN {X 0,Y 474.205,Z 571.228,A -85,B 0,C 180,E1 -7145.837,E2 -7145.837} C_VEL
LIN {X 0,Y 474.507,Z 565.407,A -85,B 0,C 180,E1 -7147.391,E2 -7147.391} C_VEL
LIN {X 0,Y 474.988,Z 557.13,A -85,B 0,C 180,E1 -7149.237,E2 -7149.237} C_VEL
LIN {X 0,Y 475.576,Z 548.514,A -85,B 0,C 180,E1 -7150.839,E2 -7150.839} C_VEL
LIN {X 0,Y 476.33,Z 538.221,A -85,B 0,C 180,E1 -7152.462,E2 -7152.462} C_VEL
LIN {X 0,Y 477.206,Z 527.158,A -85,B 0,C 180,E1 -7153.949,E2 -7153.949} C_VEL
LIN {X 0,Y 478.233,Z 514.69,A -85,B 0,C 180,E1 -7155.374,E2 -7155.374} C_VEL
LIN {X 0,Y 479.322,Z 500.879,A -85,B 0,C 180,E1 -7156.706,E2 -7156.706} C_VEL
LIN {X 0,Y 480.387,Z 486.463,A -85,B 0,C 180,E1 -7157.863,E2 -7157.863} C_VEL
LIN {X 0,Y 481.353,Z 471.995,A -85,B 0,C 180,E1 -7158.825,E2 -7158.825} C_VEL
LIN {X 0,Y 482.283,Z 456.457,A -85,B 0,C 180,E1 -7159.668,E2 -7159.668} C_VEL
LIN {X 0,Y 483.065,Z 440.098,A -85,B 0,C 180,E1 -7160.364,E2 -7160.364} C_VEL
LIN {X 0,Y 483.695,Z 424.084,A -85,B 0,C 180,E1 -7160.872,E2 -7160.872} C_VEL
LIN {X 0,Y 484.118,Z 407.747,A -85,B 0,C 180,E1 -7161.217,E2 -7161.217} C_VEL
LIN {X 0,Y 486.659,Z 229.491,A -85,B 0,C 180,E1 -7164.014,E2 -7164.014} C_VEL
LIN {X 0,Y 486.19,Z 227.119,A -85,B 0,C 180,E1 -7164.084,E2 -7164.084} C_VEL
LIN {X 0,Y 477.696,Z 208.815,A -85,B 0,C 180,E1 -7164.986,E2 -7164.986} C_VEL
LIN {X 0,Y 474.615,Z 198.678,A -85,B 0,C 180,E1 -7166.519,E2 -7166.519} C_VEL
LIN {X 0,Y 474.594,Z 198.682,A -85,B 0,C 180,E1 -7169.769,E2 -7169.769} C_VEL
LIN {X 0,Y 474.63,Z 198.676,A -85,B 0,C 180,E1 -7172.676,E2 -7172.676} C_VEL
LIN {X 0,Y 474.619,Z 198.676,A -85,B 0,C 180,E1 -7175.505,E2 -7175.505} C_VEL
LIN {X 0,Y 474.627,Z 198.678,A -85,B 0,C 180,E1 -7178.884,E2 -7178.884} C_VEL
LIN {X 0,Y 474.639,Z 198.672,A -85,B 0,C 180,E1 -7181.884,E2 -7181.884} C_VEL
LIN {X 0,Y 474.692,Z 198.664,A -85,B 0,C 180,E1 -7184.544,E2 -7184.544} C_VEL
LIN {X 0,Y 474.697,Z 198.66,A -85,B 0,C 180,E1 -7188.037,E2 -7188.037} C_VEL
LIN {X 0,Y 474.705,Z 198.663,A -85,B 0,C 180,E1 -7191.486,E2 -7191.486} C_VEL
LIN {X 0,Y 474.762,Z 198.657,A -85,B 0,C 180,E1 -7194.052,E2 -7194.052} C_VEL
LIN {X 0,Y 474.886,Z 198.64,A -85,B 0,C 180,E1 -7197.455,E2 -7197.455} C_VEL
LIN {X 0,Y 474.904,Z 198.643,A -85,B 0,C 180,E1 -7200,E2 -7200} C_VEL
LIN {X 0,Y 474.886,Z 198.642,A -85,B 0,C 180,E1 -7202.545,E2 -7202.545} C_VEL
LIN {X 0,Y 474.771,Z 198.658,A -85,B 0,C 180,E1 -7205.948,E2 -7205.948} C_VEL
LIN {X 0,Y 474.721,Z 198.663,A -85,B 0,C 180,E1 -7208.514,E2 -7208.514} C_VEL
LIN {X 0,Y 474.697,Z 198.668,A -85,B 0,C 180,E1 -7211.963,E2 -7211.963} C_VEL
LIN {X 0,Y 474.693,Z 198.667,A -85,B 0,C 180,E1 -7215.456,E2 -7215.456} C_VEL
LIN {X 0,Y 474.658,Z 198.667,A -85,B 0,C 180,E1 -7219.01,E2 -7219.01} C_VEL
LIN {X 0,Y 474.584,Z 198.682,A -85,B 0,C 180,E1 -7221.729,E2 -7221.729} C_VEL
LIN {X 0,Y 474.653,Z 198.669,A -85,B 0,C 180,E1 -7224.493,E2 -7224.493} C_VEL
LIN {X 0,Y 474.693,Z 198.667,A -85,B 0,C 180,E1 -7227.339,E2 -7227.339} C_VEL
LIN {X 0,Y 474.599,Z 198.678,A -85,B 0,C 180,E1 -7230.811,E2 -7230.811} C_VEL
LIN {X 0,Y 474.632,Z 198.676,A -85,B 0,C 180,E1 -7233.984,E2 -7233.984} C_VEL
LIN {X 0,Y 474.566,Z 198.685,A -85,B 0,C 180,E1 -7236.9,E2 -7236.9} C_VEL
LIN {X 0,Y 474.622,Z 198.679,A -85,B 0,C 180,E1 -7239.648,E2 -7239.648} C_VEL
LIN {X 0,Y 474.626,Z 198.681,A -85,B 0,C 180,E1 -7242.933,E2 -7242.933} C_VEL
LIN {X 0,Y 474.604,Z 198.68,A -85,B 0,C 180,E1 -7245.896,E2 -7245.896} C_VEL
LIN {X 0,Y 474.622,Z 198.68,A -85,B 0,C 180,E1 -7249.041,E2 -7249.041} C_VEL
LIN {X 0,Y 474.605,Z 198.678,A -85,B 0,C 180,E1 -7251.705,E2 -7251.705} C_VEL
LIN {X 0,Y 474.62,Z 198.679,A -85,B 0,C 180,E1 -7254.726,E2 -7254.726} C_VEL
LIN {X 0,Y 474.647,Z 198.757,A -85,B 0,C 180,E1 -7257.155,E2 -7257.155} C_VEL
LIN {X 0,Y 480.419,Z 217.421,A -85,B 0,C 180,E1 -7259.667,E2 -7259.667} C_VEL
LIN {X 0,Y 482.314,Z 224.041,A -85,B 0,C 180,E1 -7260.516,E2 -7260.516} C_VEL
LIN {X 0,Y 482.326,Z 228.109,A -85,B 0,C 180,E1 -7260.958,E2 -7260.958} C_VEL
LIN {X 0,Y 482.049,Z 232.043,A -85,B 0,C 180,E1 -7261.365,E2 -7261.365} C_VEL
LIN {X 0,Y 486.316,Z 256.079,A -85,B 0,C 180,E1 -7262.048,E2 -7262.048} C_VEL
LIN {X 0,Y 484.597,Z 381.833,A -85,B 0,C 180,E1 -7264.021,E2 -7264.021} C_VEL
LIN {X 0,Y 483.775,Z 440.215,A -85,B 0,C 180,E1 -7264.953,E2 -7264.953} C_VEL
LIN {X 0,Y 483.147,Z 456.303,A -85,B 0,C 180,E1 -7265.365,E2 -7265.365} C_VEL
LIN {X 0,Y 482.446,Z 471.988,A -85,B 0,C 180,E1 -7265.928,E2 -7265.928} C_VEL
LIN {X 0,Y 481.642,Z 486.103,A -85,B 0,C 180,E1 -7266.571,E2 -7266.571} C_VEL
LIN {X 0,Y 480.601,Z 502.384,A -85,B 0,C 180,E1 -7267.505,E2 -7267.505} C_VEL
LIN {X 0,Y 479.575,Z 516.605,A -85,B 0,C 180,E1 -7268.509,E2 -7268.509} C_VEL
LIN {X 0,Y 478.58,Z 529.783,A -85,B 0,C 180,E1 -7269.611,E2 -7269.611} C_VEL
LIN {X 0,Y 477.538,Z 542.843,A -85,B 0,C 180,E1 -7270.892,E2 -7270.892} C_VEL
LIN {X 0,Y 476.693,Z 554.092,A -85,B 0,C 180,E1 -7272.187,E2 -7272.187} C_VEL
LIN {X 0,Y 475.824,Z 565.714,A -85,B 0,C 180,E1 -7273.752,E2 -7273.752} C_VEL
LIN {X 0,Y 475.248,Z 575.074,A -85,B 0,C 180,E1 -7275.221,E2 -7275.221} C_VEL
LIN {X 0,Y 474.669,Z 584.492,A -85,B 0,C 180,E1 -7276.951,E2 -7276.951} C_VEL
LIN {X 0,Y 474.371,Z 591.383,A -85,B 0,C 180,E1 -7278.463,E2 -7278.463} C_VEL
LIN {X 0,Y 474.011,Z 598.06,A -85,B 0,C 180,E1 -7280.183,E2 -7280.183} C_VEL
LIN {X 0,Y 473.881,Z 603.477,A -85,B 0,C 180,E1 -7281.901,E2 -7281.901} C_VEL
LIN {X 0,Y 473.831,Z 607.722,A -85,B 0,C 180,E1 -7283.596,E2 -7283.596} C_VEL
LIN {X 0,Y 473.759,Z 610.268,A -85,B 0,C 180,E1 -7284.894,E2 -7284.894} C_VEL
LIN {X 0,Y 473.739,Z 612.771,A -85,B 0,C 180,E1 -7286.598,E2 -7286.598} C_VEL
LIN {X 0,Y 473.719,Z 614.184,A -85,B 0,C 180,E1 -7288.3,E2 -7288.3} C_VEL
LIN {X 0,Y 473.665,Z 614.719,A -85,B 0,C 180,E1 -7290,E2 -7290} C_VEL
LIN {X 0,Y 473.719,Z 614.195,A -85,B 0,C 180,E1 -7291.701,E2 -7291.701} C_VEL
LIN {X 0,Y 473.739,Z 612.792,A -85,B 0,C 180,E1 -7293.402,E2 -7293.402} C_VEL
LIN {X 0,Y 473.759,Z 610.303,A -85,B 0,C 180,E1 -7295.107,E2 -7295.107} C_VEL
LIN {X 0,Y 473.822,Z 606.877,A -85,B 0,C 180,E1 -7296.815,E2 -7296.815} C_VEL
LIN {X 0,Y 473.951,Z 601.014,A -85,B 0,C 180,E1 -7298.958,E2 -7298.958} C_VEL
LIN {X 0,Y 474.258,Z 593.3,A -85,B 0,C 180,E1 -7301.107,E2 -7301.107} C_VEL
LIN {X 0,Y 474.659,Z 585.621,A -85,B 0,C 180,E1 -7302.832,E2 -7302.832} C_VEL
LIN {X 0,Y 475.127,Z 576.443,A -85,B 0,C 180,E1 -7304.564,E2 -7304.564} C_VEL
LIN {X 0,Y 475.807,Z 566.75,A -85,B 0,C 180,E1 -7306.118,E2 -7306.118} C_VEL
LIN {X 0,Y 476.583,Z 556.007,A -85,B 0,C 180,E1 -7307.596,E2 -7307.596} C_VEL
LIN {X 0,Y 477.4,Z 544.926,A -85,B 0,C 180,E1 -7308.897,E2 -7308.897} C_VEL
LIN {X 0,Y 478.46,Z 531.255,A -85,B 0,C 180,E1 -7310.272,E2 -7310.272} C_VEL
LIN {X 0,Y 479.473,Z 518.209,A -85,B 0,C 180,E1 -7311.384,E2 -7311.384} C_VEL
LIN {X 0,Y 480.526,Z 503.596,A -85,B 0,C 180,E1 -7312.426,E2 -7312.426} C_VEL
LIN {X 0,Y 481.403,Z 490.221,A -85,B 0,C 180,E1 -7313.214,E2 -7313.214} C_VEL
LIN {X 0,Y 482.329,Z 474.684,A -85,B 0,C 180,E1 -7313.964,E2 -7313.964} C_VEL
LIN {X 0,Y 483.099,Z 459.02,A -85,B 0,C 180,E1 -7314.552,E2 -7314.552} C_VEL
LIN {X 0,Y 483.622,Z 443.253,A -85,B 0,C 180,E1 -7314.978,E2 -7314.978} C_VEL
LIN {X 0,Y 484.173,Z 420.258,A -85,B 0,C 180,E1 -7315.37,E2 -7315.37} C_VEL
LIN {X 0,Y 486.256,Z 255.942,A -85,B 0,C 180,E1 -7317.938,E2 -7317.938} C_VEL
LIN {X 0,Y 482.06,Z 232.532,A -85,B 0,C 180,E1 -7318.597,E2 -7318.597} C_VEL
LIN {X 0,Y 482.491,Z 226.005,A -85,B 0,C 180,E1 -7319.27,E2 -7319.27} C_VEL
LIN {X 0,Y 481.781,Z 222.117,A -85,B 0,C 180,E1 -7319.734,E2 -7319.734} C_VEL
LIN {X 0,Y 476.088,Z 203.426,A -85,B 0,C 180,E1 -7322.178,E2 -7322.178} C_VEL
LIN {X 0,Y 474.618,Z 198.661,A -85,B 0,C 180,E1 -7322.841,E2 -7322.841} C_VEL
LIN {X 0,Y 474.609,Z 198.677,A -85,B 0,C 180,E1 -7325.468,E2 -7325.468} C_VEL
LIN {X 0,Y 474.608,Z 198.678,A -85,B 0,C 180,E1 -7328.457,E2 -7328.457} C_VEL
LIN {X 0,Y 474.611,Z 198.676,A -85,B 0,C 180,E1 -7331.786,E2 -7331.786} C_VEL
LIN {X 0,Y 474.613,Z 198.673,A -85,B 0,C 180,E1 -7335.298,E2 -7335.298} C_VEL
LIN {X 0,Y 474.612,Z 198.676,A -85,B 0,C 180,E1 -7338.214,E2 -7338.214} C_VEL
LIN {X 0,Y 474.607,Z 198.677,A -85,B 0,C 180,E1 -7341.542,E2 -7341.542} C_VEL
LIN {X 0,Y 474.619,Z 198.673,A -85,B 0,C 180,E1 -7344.725,E2 -7344.725} C_VEL
LIN {X 0,Y 474.631,Z 198.666,A -85,B 0,C 180,E1 -7347.788,E2 -7347.788} C_VEL
LIN {X 0,Y 474.619,Z 198.68,A -85,B 0,C 180,E1 -7350.885,E2 -7350.885} C_VEL
LIN {X 0,Y 474.65,Z 198.66,A -85,B 0,C 180,E1 -7353.628,E2 -7353.628} C_VEL
LIN {X 0,Y 474.631,Z 198.678,A -85,B 0,C 180,E1 -7356.642,E2 -7356.642} C_VEL
LIN {X 0,Y 474.649,Z 198.665,A -85,B 0,C 180,E1 -7360.089,E2 -7360.089} C_VEL
LIN {X 0,Y 474.632,Z 198.675,A -85,B 0,C 180,E1 -7362.774,E2 -7362.774} C_VEL
LIN {X 0,Y 474.643,Z 198.669,A -85,B 0,C 180,E1 -7365.421,E2 -7365.421} C_VEL
LIN {X 0,Y 474.701,Z 198.652,A -85,B 0,C 180,E1 -7368.038,E2 -7368.038} C_VEL
LIN {X 0,Y 474.709,Z 198.661,A -85,B 0,C 180,E1 -7371.486,E2 -7371.486} C_VEL
LIN {X 0,Y 474.766,Z 198.658,A -85,B 0,C 180,E1 -7374.052,E2 -7374.052} C_VEL
LIN {X 0,Y 474.889,Z 198.62,A -85,B 0,C 180,E1 -7377.455,E2 -7377.455} C_VEL
LIN {X 0,Y 474.907,Z 198.636,A -85,B 0,C 180,E1 -7380,E2 -7380} C_VEL
LIN {X 0,Y 474.889,Z 198.641,A -85,B 0,C 180,E1 -7382.545,E2 -7382.545} C_VEL
LIN {X 0,Y 474.774,Z 198.647,A -85,B 0,C 180,E1 -7385.948,E2 -7385.948} C_VEL
LIN {X 0,Y 474.723,Z 198.663,A -85,B 0,C 180,E1 -7388.514,E2 -7388.514} C_VEL
